			FOR idx:=1 TO nMoverCount DO 
				nMoverInListIndex := nMoverLineDescending[nListCounter, idx];
				IF nMoverInListIndex > 0 THEN
					FOR idx2:=1 TO nMoverCount DO
						IF  MoversToSort[idx2].nMoverIndex > 0
						AND MoversToSort[idx2].nMoverIndex = nMoverInListIndex
						THEN
							IF MoversToSort[idx2].nMoverTrackOID = nTrackOID THEN
								nMoverLineCounter := nMoverLineCounter +1;
								nMoverLineDescend[nMoverLineCounter] := nMoverInListIndex;
							END_IF						
						END_IF
					END_FOR
				END_IF
			END_FOR
			
			nListCounter := nListCounter -1;
		END_WHILE
	


		
	    // Generating the ascending mover line
		FOR idx:=1 TO nMoverLineCounter DO 
			nDescendingCounter := idx;
			nAscendingCounter  := nMoverQueuCounterTotal +1-idx;
		
			IF  nAscendingCounter >  0 
			AND nAscendingCounter <= maxNumMover
			THEN
				nMoverLineAscend[nAscendingCounter] := nMoverLineDescend[nDescendingCounter];	
			ELSE
				nErrorID := -36;	
			END_IF
		END_FOR
		

	
		// Set the needed sorting direction 		
		IF nSortingDirection = eSortingDirection.ascending THEN
			nMoverLineSorted := nMoverLineAscend;
		ELSE
			nMoverLineSorted := nMoverLineDescend;
		END_IF
	
		
	    // Update mover list 
		sMoverSortedInfo := '';
		IF nMoverLineCounter = nMoverCount THEN	
			FOR idx:=1 TO nMoverLineCounter DO 
				nMoverInListIndex := nMoverLineSorted[idx];
				IF nMoverInListIndex > 0 THEN
					FOR idx2:=1 TO nMoverCount DO
						IF MoversToSort[idx2].nMoverIndex = nMoverInListIndex THEN
							MoversSorted[idx] := MoversToSort[idx2];
							 sMoverSortedInfo := CONCAT(sMoverSortedInfo, ' M');
							 sMoverSortedInfo := CONCAT(sMoverSortedInfo, UDINT_TO_STRING(MoversSorted[idx].nMoverIndex));
							EXIT;
						END_IF
					END_FOR
				END_IF		
			END_FOR
		ELSE
			nErrorID := -33;
		END_IF	

	END_IF
	

	CASE nErrorID OF
	  0:// Sorting successfully done	
		MoversList := MoversSorted;
		THIS^.ClearTrackOrder();
		      SortList := UDINT_TO_INT(nMoverLineCounter);    // Returning the number of movers sorted
		sStatusMessage := sMoverSortedInfo;	

	-31: sStatusMessage := 'Sort: No mover in list';
	-32: sStatusMessage := 'Sort: No track specified to sort on';
	-33: sStatusMessage := 'Sort: Mover found on track not specified for sorting';
	-34: sStatusMessage := 'Sort: Sorting origin bigger than length of first track';
	-35: sStatusMessage := 'Sort: Sorting origin was set to negative value';
	-36: sStatusMessage :=  CONCAT('Sort: Sorting impossible, Tracks are not consecutive! Failed at segment: ', UDINT_TO_STRING(nFailedAt));
	-37: sStatusMessage := 'Sort: Sorting not possible, check track order.';
	ELSE
		sStatusMessage := 'Sorting Error';
	END_CASE
	
	IF nErrorID < 0 THEN
		SortList := nErrorID;  // Returning the error code
	END_IF
END_METHOD

END_FUNCTION_BLOCK

// XPlanarStandardFunctions/Station/I_List
INTERFACE I_List EXTENDS __SYSTEM.IQueryInterface

{attribute 'hide'}
{attribute 'obsolete' := 'Obsolete: Please use P_SortingMode instead'}
PROPERTY P_eSortingMode : eSortingMode
GET
END_GET
SET
END_SET
END_PROPERTY

{attribute 'hide'}
{attribute 'obsolete' := 'Obsolete: Please use P_SortingOrigin instead'}
PROPERTY P_fSortingOrigin : LREAL
GET
END_GET
SET
END_SET
END_PROPERTY

{attribute 'hide'}
{attribute 'obsolete' := 'Obsolete: Please use P_NumberInList instead'}
PROPERTY P_nNumberInList : UDINT
GET
END_GET
END_PROPERTY

{attribute 'hide'}
{attribute 'obsolete' := 'Obsolete: Please use P_Result instead'}
PROPERTY P_nResult : DINT
GET
END_GET
END_PROPERTY

{attribute 'hide'}
{attribute 'obsolete' := 'Obsolete: Please use P_SortingMode instead'}
PROPERTY P_nSortingMode : INT
GET
END_GET
SET
END_SET
END_PROPERTY

{attribute 'hide'}
{attribute 'obsolete' := 'Obsolete: Please use P_Message instead'}

PROPERTY P_sMessage : STRING
GET
END_GET
END_PROPERTY

METHOD AddMover : DINT
VAR_INPUT
	ipMover		: I_XPlanarMoverStandard;
END_VAR
END_METHOD

METHOD AddTrack : DINT
VAR_INPUT
	i_Track	: I_TrackStandard;
END_VAR
END_METHOD

METHOD ClearList : BOOL
VAR_INPUT
END_VAR
END_METHOD

METHOD ClearTrackOrder : BOOL
VAR_INPUT
END_VAR
END_METHOD

METHOD GetMoverIndexInListPosition : UDINT
VAR_INPUT
	nListIndex	: UDINT;
END_VAR
END_METHOD

METHOD GetMoverInListPosition : I_XPlanarMoverStandard
VAR_INPUT
	nListPosition	: UDINT;
END_VAR
END_METHOD

PROPERTY P_FirstInList : I_XPlanarMoverStandard
GET
END_GET
END_PROPERTY

PROPERTY P_Message : STRING
GET
END_GET
END_PROPERTY

PROPERTY P_MoverList : REFERENCE TO ARRAY [1..maxNumMover] OF ST_MoverInList
GET
END_GET
END_PROPERTY


PROPERTY P_NumberInList : UDINT
GET
END_GET
END_PROPERTY

PROPERTY P_Result : DINT
GET
END_GET
END_PROPERTY

PROPERTY P_SortingMode : eSortingMode
GET
END_GET
SET
END_SET
END_PROPERTY

PROPERTY P_SortingOrigin : LREAL
GET
END_GET
SET
END_SET
END_PROPERTY

PROPERTY P_TrackBuiltInfo : ST_TrackBuiltInfo
GET
END_GET
SET
END_SET
END_PROPERTY

METHOD RemoveFirstInList : I_XPlanarMoverStandard
VAR_INPUT
END_VAR
END_METHOD

// Removes a mover from the list
METHOD RemoveFromList : DINT
VAR_INPUT
	ipMover			: I_XPlanarMoverStandard;	// Mover to remove
END_VAR
END_METHOD

METHOD SortList : INT
VAR_INPUT
END_VAR
END_METHOD

END_INTERFACE

// XPlanarStandardFunctions/Track/FB_CustomTrackIdTable
FUNCTION_BLOCK FB_CustomTrackIdTable

VAR
	CustomTrackIdTable		: ARRAY [1..Params_XPlanar.maxTrackCount] OF ST_CutomTrackID;
	nTableFillCounter		: UDINT;
END_VAR

METHOD Clear : BOOL
VAR_INPUT
END_VAR


	MEMSET(ADR(CustomTrackIdTable), 0, SIZEOF(CustomTrackIdTable));
		
	Clear := TRUE;
END_METHOD

PROPERTY P_TabelData : ARRAY [1..Params_XPlanar.maxTrackCount] OF ST_CutomTrackID;
GET
P_TabelData := CustomTrackIdTable;
END_GET
END_PROPERTY

METHOD SetTrack : int
VAR_INPUT
	TrackOID	: OTCID;
	nCustomID	: UDINT;	
END_VAR



VAR
	bTrackAlreadIn		: BOOL;
	idx					: UDINT;
END_VAR


	nTableFillCounter := nTableFillCounter +1;
	IF nTableFillCounter <= Params_XPlanar.maxTrackCount THEN
		
		bTrackAlreadIn := FALSE;
		FOR idx:=1 TO Params_XPlanar.maxTrackCount DO
			IF CustomTrackIdTable[idx].TrackOID = TrackOID THEN
				bTrackAlreadIn := TRUE;
			END_IF	
		END_FOR
	
		IF NOT bTrackAlreadIn THEN
			CustomTrackIdTable[nTableFillCounter].nCustomID := nCustomID;
			CustomTrackIdTable[nTableFillCounter].TrackOID  := TrackOID;
			SetTrack := +1;
		ELSE
			SetTrack := -1;
		END_IF
	ELSE
		SetTrack := -2;
	END_IF
END_METHOD

END_FUNCTION_BLOCK

// XPlanarStandardFunctions/Track/FB_TrackStandard
FUNCTION_BLOCK FB_TrackStandard IMPLEMENTS I_TrackStandard 
VAR_INPUT
END_VAR



VAR
	nCustomIndex			: UDINT;
	
	stTrackRef 				: MC_PlanarTrack;
	
	{attribute 'hide'}
	addToGroupCmdFb 		: MC_PlanarFeedback;
	{attribute 'hide'}
	appendLineCmdFb 		: MC_PlanarFeedback;
	{attribute 'hide'}
	appendCircleCmdFb 		: MC_PlanarFeedback;
	{attribute 'hide'}	
	appendPointCmdFb 		: MC_PlanarFeedback;
	{attribute 'hide'}
	clearCmdFb				: MC_PlanarFeedback;
	{attribute 'hide'}
	closeLoopCmdFb			: MC_PlanarFeedback;
	{attribute 'hide'}
	disableCmdFb			: MC_PlanarFeedback;
	{attribute 'hide'}
	enableCmdFb				: MC_PlanarFeedback;
	{attribute 'hide'}
	endAtTrackCmdFb			: MC_PlanarFeedback;
	{attribute 'hide'}
	removeFromGroupCmdFb	: MC_PlanarFeedback;
	{attribute 'hide'}
	startFromTrackCmdFb		: MC_PlanarFeedback;
	{attribute 'hide'}
	resetCmdFb				: MC_PlanarFeedback;
	
	{attribute 'hide'}
	endAtTrackAdvCmdFb		: MC_PlanarFeedback;
	{attribute 'hide'}
	startFromTrackAdvCmdFb	: MC_PlanarFeedback;
	{attribute 'hide'}
	appendLineAdvCmdFb 		: MC_PlanarFeedback;
	{attribute 'hide'}
	appendCircleAdvCmdFb	: MC_PlanarFeedback;
	{attribute 'hide'}
	appendPointAdvCmdFb		: MC_PlanarFeedback;
	
	
	
	stRtAddToGroup 			: ST_CommandReturn;
	stRtAppendLine 			: ST_CommandReturn;
	stRtAppendCircle		: ST_CommandReturn;
	stRtAppendPoint			: ST_CommandReturn;	
	stRtBuildTrack 			: ST_CommandReturn;
	stRtBuildTrackExt 		: ST_CommandReturn;
	stRtBuildTrackAdv 		: ST_CommandReturn;		
	stRtClear				: ST_CommandReturn;
	stRtCloseLoop			: ST_CommandReturn;
	stRtDiable				: ST_CommandReturn;
	stRtEnable				: ST_CommandReturn;
	stRtEndAtTrack			: ST_CommandReturn;
	stRtRemoveFromGroup 	: ST_CommandReturn; 
	stRtStartFromTrack		: ST_CommandReturn;
	stRtReset				: ST_CommandReturn;

	stRtAppendLineAdv 		: ST_CommandReturn;
	stRtAppendCircleAdv		: ST_CommandReturn;
	stRtAppendPointAdv		: ST_CommandReturn;
	stRtEndAtTrackAdv		: ST_CommandReturn;
	stRtStartFromTrackAdv	: ST_CommandReturn;

	

	{attribute 'hide'}
	eState 							: E_MethodKeepAliveTrack;	
	{attribute 'hide'}
	nState							: INT;
	{attribute 'hide'}
	Busy 							: BOOL;
	{attribute 'hide'}
	_bTrackCheck					: BOOL;
	{attribute 'hide'}
	_TrackTableExt					: ARRAY[1..maxNumTrackPoints] OF ST_TrackTable;
	{attribute 'hide'}
	_TrackTableAdv					: ARRAY[1..maxNumTrackPoints] OF ST_TrackTable;
	{attribute 'hide'}
	_TrackTable						: ARRAY [1..maxNumTrackPoints,1..3] OF LREAL;
	//{attribute 'hide'}
	_startFromTrackOptions			: ST_StartFromTrackAdvancedOptions;
	//{attribute 'hide'}
	_endAtTrackOptions				: ST_EndAtTrackAdvancedOptions;
	//{attribute 'hide'}
	_ipStartFromTrack				: I_TrackStandard;	
	//{attribute 'hide'}	
	_ipEndAtTrack 					: I_TrackStandard;
	{attribute 'hide'}
	_bCloseLoop						: BOOL;	
	{attribute 'hide'}
	_nTrackBuilderErrorSituation	: UDINT;
	{attribute 'hide'}
	sBuildTrackExtInfoText			: STRING;
	{attribute 'hide'}
	sBuildTrackAdvInfoText			: STRING;
	{attribute 'hide'}
	nStateBuildTrackAdvanced 		: INT;
	
	// logging
	{attribute 'hide'}
	stTimeZoneInfo 				: TC2_UTILITIES.ST_TimeZoneInformation; //all times are UTC and must be converted to local time zone. if no timezone given only UTC times are avaialbe		
	{attribute 'hide'}
	_eLogSeverity				: TcEventSeverity := TcEventSeverity.VERBOSE;
	{attribute 'hide'}
	stLastCommand				: ST_TrackCommand;	
	aLog						: ARRAY[0..MAX_LAST_LOGS] OF ST_TrackCommandLog;
	
END_VAR


VAR_STAT
	{attribute 'hide'}	
	nTrackBuiltCountInfo	: UDINT;
	{attribute 'hide'}
	nTrackBuiltCount		: UDINT;
	{attribute 'hide'}
	TrackInfo				: ARRAY[1..maxTrackCount] OF ST_TrackInfo;	
	{attribute 'hide'}
	nTrackBuiltTable		: ARRAY[1..maxTrackCount] OF UDINT;
END_VAR

{attribute 'hide'}
METHOD PROTECTED ccl_BuildTrack : BOOL

VAR_INST
	TrackTableInt		: ARRAY [1..maxNumTrackPoints,1..3] OF LREAL;		
	nState				: INT;
	fbR_TrigExecute 	: R_TRIG;
	bCloseLoopFlag		: BOOL;
	nPointIndex			: INT;
	nPointIndexA		: INT;	
	nPointIndexB		: INT;	
	fTestValue			: LREAL;
	idx1, idx2			: INT;
	trackLinePosStart 	: PositionXYC;
	trackLinePosEnd 	: PositionXYC;
END_VAR
CASE nState OF 
	
	0:	// Init
		stRtBuildTrack.Done := FALSE;
		stRtBuildTrack.Busy := TRUE;
		  TrackTableInt := _TrackTable;
	     bCloseLoopFlag := _bCloseLoop;
		    nPointIndex := -1;
		         nState := 100;
	
		
	100: // Building the track
		IF nPointIndex = -1 THEN
			IF _ipStartFromTrack <> 0 THEN
				nState := 110;
			END_IF
			nPointIndex := 0;
		ELSE
			IF nPointIndex < UINT_TO_INT(maxNumTrackPoints-1) THEN
				IF nPointIndex = 0 THEN
					nPointIndex := 1;
				ELSE
					nPointIndex := nPointIndex + 2;
				END_IF
				
				nPointIndexA := nPointIndex;
				nPointIndexB := nPointIndex +1;
				
				fTestValue := 0;
				FOR idx1:=nPointIndexA TO nPointIndexB DO 
					FOR idx2 := 1 TO 3 DO
						fTestValue := fTestValue + _TrackTable[idx1,idx2];	
					END_FOR
				END_FOR
				
				IF fTestValue > 0 THEN
					nState := 120;
				ELSE
					IF _ipEndAtTrack <> 0 THEN
						nPointIndex := UINT_TO_INT(maxNumTrackPoints);
						     nState := 130;
					ELSE
						nPointIndex := UINT_TO_INT(maxNumTrackPoints);
					END_IF
				END_IF
		
			ELSE
				IF bCloseLoopFlag THEN
					nState := 140;
				ELSE
					nState := 200;
				END_IF	
			END_IF
		END_IF
	
	
	110:  // When starting from another track
			IF _ipStartFromTrack <> 0 THEN
			THIS^.StartFromTrack(_ipStartFromTrack);
			nState := 111;
			END_IF
			
	111: 	
			IF startFromTrackCmdFb.Done THEN
				nState := 100;
			END_IF

	120: // Append Line
			trackLinePosStart.SetValuesXYC( _TrackTable[nPointIndexA,1], _TrackTable[nPointIndexA,2], _TrackTable[nPointIndexA,3]);
			trackLinePosEnd.SetValuesXYC(   _TrackTable[nPointIndexB,1], _TrackTable[nPointIndexB,2], _TrackTable[nPointIndexB,3]);
			THIS^.AppendLine(trackLinePosStart,trackLinePosEnd);
			nState := 121;			
			
	121: 
			IF appendLineCmdFb.Done THEN
				nState := 100;
			END_IF	
			
			
	130:  // When ending at another track
			IF _ipEndAtTrack <> 0 THEN
			THIS^.EndAtTrack(_ipEndAtTrack); 
				nState := 131;
			END_IF
			
	131: 
			IF endAtTrackCmdFb.Done THEN
				nState := 100;
			END_IF		
		
	140:  // Closing the track 
			bCloseLoopFlag := FALSE;
			stTrackRef.CloseLoop(closeLoopCmdFb);
			nState := 141;	
			
	141:
			IF closeLoopCmdFb.Done THEN
				nState := 100;
			END_IF
			
			 
	200: 	// MC_Reset Done
			eState 					:= E_MethodKeepAliveTrack.eIdle; 
			nState 					:= 0;
			stRtBuildTrack.Done 	:= TRUE;
			stRtBuildTrack.Busy 	:= FALSE;
			stRtBuildTrack.Active 	:= FALSE;
			ccl_BuildTrack 			:= TRUE;

END_CASE
END_METHOD

//{attribute 'hide'}
METHOD PROTECTED ccl_BuildTrackAdv : BOOL

VAR_INST
	TrackTableInt		: ARRAY[1..maxNumTrackPoints] OF ST_TrackTable;		
	nState				: INT;
	fbR_TrigExecute 	: R_TRIG;
	bCloseLoopFlag		: BOOL;
	nPointIndex			: UINT;

	trackPos 			: PositionXYC;
	trackPosStart 		: PositionXYC;
	trackPosEnd 		: PositionXYC;
	trackPosRef 		: PositionXYC;
	trackPosStartRef 	: PositionXYC;
	trackPosEndRef 		: PositionXYC;	
	trackPosCenter		: PositionXY;

	nErrorId			: UDINT;	
	nErrorSituation		: UDINT;
	
	nTrackOID			: UDINT;

	idx						: UDINT;
	bPreceedingTrackExists	: BOOL;
	bFollowingTrackExists	: BOOL;
	
	bClockWise	: BOOL;
END_VAR


VAR
	stCommand : ST_TrackCommand;
END_VAR
CASE nState OF 
	

	0:	// Init
		stRtBuildTrackAdv.Active := TRUE;
		stRtBuildTrackAdv.Busy   := TRUE;
		stRtBuildTrackAdv.Done   := FALSE;
		
		   TrackTableInt := _TrackTableAdv;
	      bCloseLoopFlag := _bCloseLoop;
		  	    nErrorId := 0;
		 nErrorSituation := 0;
		     nPointIndex := 0;
		          nState := 10;
				 
				 
	10:	// Check if track table is plausible
		IF _bTrackCheck THEN
			nState := 20;
		ELSE
			nErrorSituation := 1;
			nState := 950;
		END_IF			 
				
 
	20: // Check if track is linked to hardware
		nTrackOID := THIS^.P_OID;	
		IF nTrackOID > 0 THEN
			nState := nState + 10;
		ELSE
			nErrorSituation := 8;
			nState := 950;				
		END_IF	
		
		
	30: // Check if the preceding track exists
		bPreceedingTrackExists := FALSE;
		IF _ipStartFromTrack <> 0 THEN	
			FOR idx:=1 TO maxTrackCount DO 
				IF nTrackBuiltTable[idx] = _ipStartFromTrack.P_OID  THEN
					bPreceedingTrackExists := TRUE;
					EXIT;	
				END_IF
			END_FOR
			
			IF bPreceedingTrackExists THEN
				nState := nState + 10;
			ELSE
				nErrorSituation := 9;
				nState := 950;						
			END_IF	
		ELSE
			nState := nState + 10;
		END_IF
		
		
	40: // Check if the following track exists
		bFollowingTrackExists := FALSE;
		IF _ipEndAtTrack <> 0 THEN	
			FOR idx:=1 TO maxTrackCount DO 
				IF nTrackBuiltTable[idx] = _ipEndAtTrack.P_OID  THEN
					bFollowingTrackExists := TRUE;
					EXIT;	
				END_IF
			END_FOR
			
			IF bFollowingTrackExists THEN
				nState := nState + 10;
			ELSE
				nErrorSituation := 10;
				nState := 950;						
			END_IF	
		ELSE
			nState := nState + 10;
		END_IF		
		
		
	50:	nState := 100;
	
	
		 	 
	100: 	// Building the track
			IF nPointIndex = 0 THEN
				nPointIndex := 1;
				IF _ipStartFromTrack <> 0 THEN
					nState := 110;
				END_IF
			ELSE
				IF nPointIndex < maxNumTrackPoints THEN
					
					IF TrackTableInt[nPointIndex].ePointType = E_PointType.Point THEN
						nState := 200;		
					ELSIF TrackTableInt[nPointIndex].ePointType = E_PointType.Line_Start THEN
						nState := 300;
					ELSIF TrackTableInt[nPointIndex].ePointType = E_PointType.Circle_Start THEN
						nState := 400;	
					ELSIF TrackTableInt[nPointIndex].ePointType = E_PointType.none THEN
						nState := 500;	
					END_IF
					
				END_IF
			END_IF
		
	
	110:  // When starting from another track
			IF TrackTableInt[nPointIndex].ReferenceSystem = 0 THEN
				nState := 120;
			ELSE
				nState := 130;
			END_IF	
	
	120:	// Starting from another track without reference system
			IF _ipStartFromTrack <> 0 THEN
			THIS^.StartFromTrack(_ipStartFromTrack);     
				nState := nState +1;
			END_IF
			
	121: 	IF startFromTrackCmdFb.Done THEN
				nState := 100;
			ELSIF startFromTrackCmdFb.Error THEN
				       nErrorId := startFromTrackCmdFb.ErrorId;
				nErrorSituation := 2;
				nState := 950;				
			END_IF	
	
			
	130:	// Starting from another track with reference system
			IF _ipStartFromTrack <> 0 THEN
			THIS^.StartFromTrackAdv(_ipStartFromTrack, _startFromTrackOptions);     
				nState := nState +1;
			END_IF
			
	131: 	
			IF startFromTrackAdvCmdFb.Done THEN
				nState := 100;
			ELSIF startFromTrackAdvCmdFb.Error THEN
				       nErrorId := startFromTrackAdvCmdFb.ErrorId;
				nErrorSituation := 2;
				nState := 950;				
			END_IF
			



	200:	// Append Point
			IF TrackTableInt[nPointIndex].ReferenceSystem = 0 THEN
				nState := 210;
			ELSE
				nState := 220;
			END_IF

			
	210:	// Append Point without reference system
			trackPos.SetValuesXYC(TrackTableInt[nPointIndex].fPointPosition_X, TrackTableInt[nPointIndex].fPointPosition_Y,  TrackTableInt[nPointIndex].fPointOrientation_C);
	
			THIS^.AppendPoint(trackPosRef);
			nPointIndex := nPointIndex +1;
			nState := nState + 11;	
			
	211:	IF appendPointCmdFb.Done THEN
				nState := 100;
			ELSIF appendPointCmdFb.Error THEN
				       nErrorId := appendPointCmdFb.ErrorId;
				nErrorSituation := 3;
				nState := 950;				
			END_IF			
			
			
	220:	// Append Point with reference system
			trackPosRef.SetValuesXYC(TrackTableInt[nPointIndex].fPointPosition_X, TrackTableInt[nPointIndex].fPointPosition_Y,  TrackTableInt[nPointIndex].fPointOrientation_C);
			trackPosRef.ReferenceId := TrackTableInt[nPointIndex].ReferenceSystem;
	
			THIS^.AppendPoint(trackPosRef);
			nPointIndex := nPointIndex +1;
			nState := nState + 11;	
			
	221:	IF appendPointCmdFb.Done THEN
				nState := 100;
			ELSIF appendPointCmdFb.Error THEN
				       nErrorId := appendPointCmdFb.ErrorId;
				nErrorSituation := 3;
				nState := 950;				
			END_IF


			
	300:	// Append Line
			IF TrackTableInt[nPointIndex].ReferenceSystem = 0 THEN
				nState := 310;
			ELSE
				nState := 320;
			END_IF

	310:	// Adding the line without reference system
			trackPosStart.SetValuesXYC(TrackTableInt[nPointIndex].fPointPosition_X, TrackTableInt[nPointIndex].fPointPosition_Y,  TrackTableInt[nPointIndex].fPointOrientation_C);
			trackPosEnd.SetValuesXYC(TrackTableInt[nPointIndex+1].fPointPosition_X, TrackTableInt[nPointIndex+1].fPointPosition_Y,  TrackTableInt[nPointIndex+1].fPointOrientation_C);
			
			THIS^.AppendLine(trackPosStart,trackPosEnd);
			nState := nState + 1;	
			
	311:	IF appendLineCmdFb.Done THEN
				nPointIndex := nPointIndex +2;
				nState := 100;
			ELSIF appendLineCmdFb.Error THEN
				       nErrorId := appendLineCmdFb.ErrorId;
				nErrorSituation := 4;
				nState := 950;				
			END_IF	

			
	320:	// Adding the line with reference system
			trackPosStartRef.SetValuesXYC(TrackTableInt[nPointIndex].fPointPosition_X, TrackTableInt[nPointIndex].fPointPosition_Y,  TrackTableInt[nPointIndex].fPointOrientation_C);
			trackPosEndRef.SetValuesXYC(TrackTableInt[nPointIndex+1].fPointPosition_X, TrackTableInt[nPointIndex+1].fPointPosition_Y,  TrackTableInt[nPointIndex+1].fPointOrientation_C);
			
			trackPosStartRef.ReferenceId := TrackTableInt[nPointIndex].ReferenceSystem;
			trackPosEndRef.ReferenceId   := TrackTableInt[nPointIndex+1].ReferenceSystem;

			THIS^.AppendLine(trackPosStartRef,trackPosEndRef);
			
			nState := nState + 1;	
			
	321:	IF appendLineCmdFb.Done THEN
				nPointIndex := nPointIndex +2;
				nState := 100;
			ELSIF appendLineCmdFb.Error THEN
				       nErrorId := appendLineCmdFb.ErrorId;
				nErrorSituation := 4;
				nState := 950;				
			END_IF		
			

			
	400:	// Append Circle
			IF TrackTableInt[nPointIndex].ReferenceSystem = 0 THEN
				nState := 410;
			ELSE
				nState := 420;
			END_IF
			
	410:	// Append Circle without reference system
			trackPosStart.SetValuesXYC( TrackTableInt[nPointIndex+0].fPointPosition_X,  TrackTableInt[nPointIndex+0].fPointPosition_Y,    TrackTableInt[nPointIndex+0].fPointOrientation_C);
			trackPosCenter.SetValuesXY( TrackTableInt[nPointIndex+1].fPointPosition_X,  TrackTableInt[nPointIndex+1].fPointPosition_Y );
			trackPosEnd.SetValuesXYC(   TrackTableInt[nPointIndex+2].fPointPosition_X,  TrackTableInt[nPointIndex+2].fPointPosition_Y,    TrackTableInt[nPointIndex+2].fPointOrientation_C);
			
			bClockWise := FALSE;
			CASE TrackTableInt[nPointIndex+1].eOption OF
			E_PointOption.Circle_Clockwise: 		bClockWise := TRUE;			
			E_PointOption.Circle_CounterClockwise:	bClockWise := FALSE;		
			END_CASE

			THIS^.AppendCircle(trackPosStart,trackPosCenter,trackPosEnd, bClockWise);
			nPointIndex := nPointIndex +3;
			nState := nState + 10;	
			
	411:	IF appendCircleCmdFb.Done THEN
				nState := 100;
			ELSIF appendCircleCmdFb.Error THEN
				       nErrorId := appendCircleCmdFb.ErrorId;
				nErrorSituation := 5;
				nState := 950;				
			END_IF	


	420:	// Append Circle with reference system
			trackPosStartRef.SetValuesXYC( TrackTableInt[nPointIndex+0].fPointPosition_X,  TrackTableInt[nPointIndex+0].fPointPosition_Y,    TrackTableInt[nPointIndex+0].fPointOrientation_C);
			trackPosCenter.SetValuesXY( TrackTableInt[nPointIndex+1].fPointPosition_X,  TrackTableInt[nPointIndex+1].fPointPosition_Y );
			trackPosEndRef.SetValuesXYC(   TrackTableInt[nPointIndex+2].fPointPosition_X,  TrackTableInt[nPointIndex+2].fPointPosition_Y,    TrackTableInt[nPointIndex+2].fPointOrientation_C);

			trackPosStartRef.ReferenceId := TrackTableInt[nPointIndex].ReferenceSystem;
			trackPosEndRef.ReferenceId   := TrackTableInt[nPointIndex+2].ReferenceSystem;			
			
			bClockWise := FALSE;
			CASE TrackTableInt[nPointIndex+1].eOption OF
			E_PointOption.Circle_Clockwise: 		bClockWise := TRUE;			
			E_PointOption.Circle_CounterClockwise:	bClockWise := FALSE;		
			END_CASE

			THIS^.AppendCircle(trackPosStartRef,trackPosCenter,trackPosEndRef, bClockWise);
			nPointIndex := nPointIndex +3;
			nState := nState + 1;	
			
	421:	
			appendCircleCmdFb.Update();
			IF appendCircleCmdFb.Done THEN
				nState := 100;
			ELSIF appendCircleCmdFb.Error THEN
				       nErrorId := appendCircleCmdFb.ErrorId;
				nErrorSituation := 5;
				nState := 950;				
			END_IF	


			
	500:	// Check if this track is ending on another track  
			IF _ipEndAtTrack <> 0 THEN
				nState := nState + 10;	
			ELSE
				nState := 600;
			END_IF			
			
					
	510:  	// Check if this track has a reference system
			IF TrackTableInt[nPointIndex-1].ReferenceSystem = 1 THEN
				nState := 520;
			ELSE
				nState := 530;
			END_IF				
			

	520:	THIS^.EndAtTrackAdv(_ipEndAtTrack, _endAtTrackOptions); 
			nState := nState + 1;	
		
	521:	IF endAtTrackAdvCmdFb.Done THEN
				nState := 900;
			ELSIF endAtTrackAdvCmdFb.Error THEN
				       nErrorId := endAtTrackAdvCmdFb.ErrorId;
				nErrorSituation := 6;
				nState := 950;				
			END_IF		

			
	530:	THIS^.EndAtTrack(_ipEndAtTrack); 
			nState := nState + 1;	
		
	531:	IF endAtTrackCmdFb.Done THEN
				nState := 900;
			ELSIF endAtTrackCmdFb.Error THEN
				       nErrorId := endAtTrackAdvCmdFb.ErrorId;
				nErrorSituation := 6;
				nState := 950;				
			END_IF					
			
			
	600:	// Check if this track closes the loop
			IF bCloseLoopFlag THEN
				THIS^.CloseLoop();
				nState := nState + 10;
			ELSE
				nState := nState + 100;
			END_IF
			
	610:	IF closeLoopCmdFb.Done THEN
				nState := nState + 90;
			ELSIF closeLoopCmdFb.Error THEN
				       nErrorId := closeLoopCmdFb.ErrorId;
				nErrorSituation := 7;
				nState := 950;				
			END_IF		
			
			
	700:	nState := 900;			
			
				 
	900: 	// BuildTrack successfully done	
			_nTrackBuilderErrorSituation := nErrorSituation;

			nTrackBuiltCount := nTrackBuiltCount +1;
			nTrackBuiltTable[nTrackBuiltCount] := THIS^.P_OID;
				
			stRtBuildTrackAdv.Done 		:= TRUE;
			stRtBuildTrackAdv.Busy 		:= FALSE;
			stRtBuildTrackAdv.Active 	:= FALSE;
			stRtBuildTrackAdv.Error     := FALSE;
			stRtBuildTrackAdv.ErrorID   := nErrorId;
			nState := 1000;
			
			
	950:	// In case of an error
			_nTrackBuilderErrorSituation := nErrorSituation;
 
			stRtBuildTrackAdv.Done 		:= FALSE;
			stRtBuildTrackAdv.Busy 		:= FALSE;
			stRtBuildTrackAdv.Active 	:= FALSE;
			stRtBuildTrackAdv.Error     := TRUE;
			stRtBuildTrackAdv.ErrorID   := nErrorId;
			nState := 1000;
			
			
	1000:	// Done
			CASE _nTrackBuilderErrorSituation OF
			 0:	sBuildTrackAdvInfoText := 'NoError';
			 1:	sBuildTrackAdvInfoText := 'TrackTableNotPlausible';	
			 2:	sBuildTrackAdvInfoText := 'StartFromTrackFailed';	
			 3:	sBuildTrackAdvInfoText := 'AppendPointFailed';
			 4:	sBuildTrackAdvInfoText := 'AppendLineFailed';
			 5:	sBuildTrackAdvInfoText := 'AppendCircleFailed';	
			 6:	sBuildTrackAdvInfoText := 'EndAtTrackFailed';	
			 7:	sBuildTrackAdvInfoText := 'CloseLoopFailed';
			 8:	sBuildTrackAdvInfoText := 'NotLinkedToNC';
			 9: sBuildTrackAdvInfoText := 'Preceeding track needs to be built first!';
			10: sBuildTrackAdvInfoText := 'Following track needs to be built first!';
			END_CASE

			ccl_BuildTrackAdv 	:= TRUE;	
			eState 				:= E_MethodKeepAliveTrack.eIdle; 
			nState 				:= 0;			
			
			
			// Update Command History
			stCommand.eCommandType 				  := eTrackCommand_eBuildTrack;
			stCommand.stBuildTrack.bSuccess 	  := stRtBuildTrackAdv.Done;
			stCommand.stBuildTrack.fTrackLength   := stTrackRef.GetLength();
			stCommand.stBuildTrack.bError 		  := stRtBuildTrackAdv.Error;
			stCommand.stBuildTrack.nErrorCode	  := stRtBuildTrackAdv.ErrorID;
			stCommand.stBuildTrack.sBuildInfoText := sBuildTrackAdvInfoText;
			UpdateCommandHistory(stCommand);

END_CASE

nStateBuildTrackAdvanced := nState;
END_METHOD

//{attribute 'hide'}
METHOD PROTECTED ccl_BuildTrackExt : BOOL

VAR_INST
	TrackTableInt		: ARRAY[1..maxNumTrackPoints] OF ST_TrackTable;;		
	nState				: INT;
	fbR_TrigExecute 	: R_TRIG;
	bCloseLoopFlag		: BOOL;
	nPointIndex			: UINT;

	trackPos 			: PositionXYC;
	trackPosStart 		: PositionXYC;
	trackPosEnd 		: PositionXYC;
	trackPosCenter		: PositionXY;

	nErrorId			: UDINT;	
	nErrorSituation		: UDINT;
	
	nTrackOID			: UDINT;

	idx						: UDINT;
	bPreceedingTrackExists	: BOOL;
	bFollowingTrackExists	: BOOL;
	
	bClockWise	: BOOL;
END_VAR


VAR
	stCommand : ST_TrackCommand;
END_VAR
CASE nState OF 
	

	0:	// Init
		stRtBuildTrackExt.Active := TRUE;
		stRtBuildTrackExt.Busy   := TRUE;
		stRtBuildTrackExt.Done   := FALSE;
		
		   TrackTableInt := _TrackTableExt;
	      bCloseLoopFlag := _bCloseLoop;
		  	    nErrorId := 0;
		 nErrorSituation := 0;
		     nPointIndex := 0;
		          nState := 10;
				 
				 
	10:	// Check if track table is plausible
		IF _bTrackCheck THEN
			nState := 20;
		ELSE
			nErrorSituation := 1;
			nState := 950;
		END_IF			 
				
 
	20: // Check if track is linked to hardware
		nTrackOID := THIS^.P_OID;	
		IF nTrackOID > 0 THEN
			nState := nState + 10;
		ELSE
			nErrorSituation := 8;
			nState := 950;				
		END_IF	
		
		
	30: // Check if the preceding track exists
		bPreceedingTrackExists := FALSE;
		IF _ipStartFromTrack <> 0 THEN	
			FOR idx:=1 TO maxTrackCount DO 
				IF nTrackBuiltTable[idx] = _ipStartFromTrack.P_OID  THEN
					bPreceedingTrackExists := TRUE;
					EXIT;	
				END_IF
			END_FOR
			
			IF bPreceedingTrackExists THEN
				nState := nState + 10;
			ELSE
				nErrorSituation := 9;
				nState := 950;						
			END_IF	
		ELSE
			nState := nState + 10;
		END_IF
		
		
	40: // Check if the following track exists
		bFollowingTrackExists := FALSE;
		IF _ipEndAtTrack <> 0 THEN	
			FOR idx:=1 TO maxTrackCount DO 
				IF nTrackBuiltTable[idx] = _ipEndAtTrack.P_OID  THEN
					bFollowingTrackExists := TRUE;
					EXIT;	
				END_IF
			END_FOR
			
			IF bFollowingTrackExists THEN
				nState := nState + 10;
			ELSE
				nErrorSituation := 10;
				nState := 950;						
			END_IF	
		ELSE
			nState := nState + 10;
		END_IF		
		
		
	50:	nState := 100;
	
	
		 	 
	100: 	// Building the track
			IF nPointIndex = 0 THEN
				IF _ipStartFromTrack <> 0 THEN
					nState := 110;
				END_IF
				nPointIndex := 1;
			ELSE
				IF nPointIndex < maxNumTrackPoints THEN
					
					IF TrackTableInt[nPointIndex].ePointType = E_PointType.Point THEN
						nState := 200;		
					ELSIF TrackTableInt[nPointIndex].ePointType = E_PointType.Line_Start THEN
						nState := 300;
					ELSIF TrackTableInt[nPointIndex].ePointType = E_PointType.Circle_Start THEN
						nState := 400;	
					ELSIF TrackTableInt[nPointIndex].ePointType = E_PointType.none THEN
						nState := 500;	
					END_IF
					
				END_IF
			END_IF
		
	
	110:  // When starting from another track
			IF _ipStartFromTrack <> 0 THEN
			THIS^.StartFromTrack(_ipStartFromTrack);
			nState := 111;
			END_IF
			
	111: 	
			IF startFromTrackCmdFb.Done THEN
				nState := 100;
			ELSIF startFromTrackCmdFb.Error THEN
				       nErrorId := startFromTrackCmdFb.ErrorId;
				nErrorSituation := 2;
				nState := 950;				
			END_IF
			
			
			
	200:	// Append Point
			trackPos.SetValuesXYC(TrackTableInt[nPointIndex].fPointPosition_X, TrackTableInt[nPointIndex].fPointPosition_Y,  TrackTableInt[nPointIndex].fPointOrientation_C);
			THIS^.AppendPoint(trackPos);
			nPointIndex := nPointIndex +1;
			nState := nState + 10;	
			
	210:	IF appendPointCmdFb.Done THEN
				nState := 100;
			ELSIF appendPointCmdFb.Error THEN
				       nErrorId := appendPointCmdFb.ErrorId;
				nErrorSituation := 3;
				nState := 950;				
			END_IF


			
	300:	// Append Line
			trackPosStart.SetValuesXYC(TrackTableInt[nPointIndex].fPointPosition_X, TrackTableInt[nPointIndex].fPointPosition_Y,  TrackTableInt[nPointIndex].fPointOrientation_C);
			trackPosEnd.SetValuesXYC(TrackTableInt[nPointIndex+1].fPointPosition_X, TrackTableInt[nPointIndex+1].fPointPosition_Y,  TrackTableInt[nPointIndex+1].fPointOrientation_C);
			THIS^.AppendLine(trackPosStart,trackPosEnd);
			nPointIndex := nPointIndex +2;
			nState := nState + 10;	
			
	310:	IF appendLineCmdFb.Done THEN
				nState := 100;
			ELSIF appendLineCmdFb.Error THEN
				       nErrorId := appendLineCmdFb.ErrorId;
				nErrorSituation := 4;
				nState := 950;				
			END_IF		
			
			
	400:	// Append Circle
			trackPosStart.SetValuesXYC( TrackTableInt[nPointIndex+0].fPointPosition_X,  TrackTableInt[nPointIndex+0].fPointPosition_Y,    TrackTableInt[nPointIndex+0].fPointOrientation_C);
			trackPosCenter.SetValuesXY( TrackTableInt[nPointIndex+1].fPointPosition_X,  TrackTableInt[nPointIndex+1].fPointPosition_Y );
			trackPosEnd.SetValuesXYC(   TrackTableInt[nPointIndex+2].fPointPosition_X,  TrackTableInt[nPointIndex+2].fPointPosition_Y,    TrackTableInt[nPointIndex+2].fPointOrientation_C);

			bClockWise := FALSE;
			CASE TrackTableInt[nPointIndex+1].eOption OF
			E_PointOption.Circle_Clockwise: 		bClockWise := TRUE;			
			E_PointOption.Circle_CounterClockwise:	bClockWise := FALSE;		
			END_CASE

			THIS^.AppendCircle(trackPosStart,trackPosCenter,trackPosEnd, bClockWise);
			nPointIndex := nPointIndex +3;
			nState := nState + 10;	
			
	410:	IF appendCircleCmdFb.Done THEN
				nState := 100;
			ELSIF appendCircleCmdFb.Error THEN
				       nErrorId := appendCircleCmdFb.ErrorId;
				nErrorSituation := 5;
				nState := 950;				
			END_IF	


	500:	// Check if this track is ending on another track 
			IF _ipEndAtTrack <> 0 THEN
				THIS^.EndAtTrack(_ipEndAtTrack); 
				nState := nState + 10;	
			ELSE
				nState := 600;
			END_IF
	
	510:	IF endAtTrackCmdFb.Done THEN
				nState := 900;
			ELSIF endAtTrackCmdFb.Error THEN
				       nErrorId := endAtTrackCmdFb.ErrorId;
				nErrorSituation := 6;
				nState := 950;				
			END_IF		

			
	600:	// Check if this track closes the loop
			IF bCloseLoopFlag THEN
				THIS^.CloseLoop();
				nState := nState + 10;
			ELSE
				nState := nState + 100;
			END_IF
			
	610:	IF closeLoopCmdFb.Done THEN
				nState := nState + 90;
			ELSIF closeLoopCmdFb.Error THEN
				       nErrorId := closeLoopCmdFb.ErrorId;
				nErrorSituation := 7;
				nState := 950;				
			END_IF		
			
			
	700:	nState := 900;			
			
				 
	900: 	// BuildTrack successfully done	
			_nTrackBuilderErrorSituation := nErrorSituation;

			nTrackBuiltCount := nTrackBuiltCount +1;
			nTrackBuiltTable[nTrackBuiltCount] := THIS^.P_OID;
				
			stRtBuildTrackExt.Done 		:= TRUE;
			stRtBuildTrackExt.Busy 		:= FALSE;
			stRtBuildTrackExt.Active 	:= FALSE;
			stRtBuildTrackExt.Error     := FALSE;
			stRtBuildTrackExt.ErrorID   := nErrorId;
			nState := 1000;
			
			
	950:	// In case of an error
			_nTrackBuilderErrorSituation := nErrorSituation;
 
			stRtBuildTrackExt.Done 		:= FALSE;
			stRtBuildTrackExt.Busy 		:= FALSE;
			stRtBuildTrackExt.Active 	:= FALSE;
			stRtBuildTrackExt.Error     := TRUE;
			stRtBuildTrackExt.ErrorID   := nErrorId;
			nState := 1000;
			
			
	1000:	// Done
			CASE _nTrackBuilderErrorSituation OF
			 0:	sBuildTrackExtInfoText := 'NoError';
			 1:	sBuildTrackExtInfoText := 'TrackTableNotPlausible';	
			 2:	sBuildTrackExtInfoText := 'StartFromTrackFailed';	
			 3:	sBuildTrackExtInfoText := 'AppendPointFailed';
			 4:	sBuildTrackExtInfoText := 'AppendLineFailed';
			 5:	sBuildTrackExtInfoText := 'AppendCircleFailed';	
			 6:	sBuildTrackExtInfoText := 'EndAtTrackFailed';	
			 7:	sBuildTrackExtInfoText := 'CloseLoopFailed';
			 8:	sBuildTrackExtInfoText := 'NotLinkedToNC';
			 9: sBuildTrackExtInfoText := 'Preceeding track needs to be built first!';
			10: sBuildTrackExtInfoText := 'Following track needs to be built first!';
			END_CASE

			ccl_BuildTrackExt 	:= TRUE;	
			eState 				:= E_MethodKeepAliveTrack.eIdle; 
			nState 				:= 0;			
			
			// Update Command History
			stCommand.eCommandType 				  := eTrackCommand_eBuildTrack;
			stCommand.stBuildTrack.bSuccess 	  := stRtBuildTrackExt.Done;
			stCommand.stBuildTrack.fTrackLength   := stTrackRef.GetLength();
			stCommand.stBuildTrack.bError 		  := stRtBuildTrackExt.Error;
			stCommand.stBuildTrack.nErrorCode	  := stRtBuildTrackExt.ErrorID;
			stCommand.stBuildTrack.sBuildInfoText := sBuildTrackExtInfoText;
			UpdateCommandHistory(stCommand);

END_CASE
END_METHOD

{attribute 'hide'}
METHOD PROTECTED ccl_MethodKeepAlive : BOOL
VAR_INPUT
END_VAR
VAR_INST

END_VAR
CASE eState OF
	
	E_MethodKeepAliveTrack.eIdle:
		nState := 0;
	
	E_MethodKeepAliveTrack.eBuildTrack:
		ccl_BuildTrack();	
		
	E_MethodKeepAliveTrack.eBuildTrackExt:
		ccl_BuildTrackExt();	

	E_MethodKeepAliveTrack.eBuildTrackAdv:
		ccl_BuildTrackAdv();					

	E_MethodKeepAliveTrack.eError:
		;
		
END_CASE
END_METHOD

{attribute 'hide'}
METHOD PROTECTED CopyReturnStructure : ST_CommandReturn
VAR_INPUT
	mcInStructur : REFERENCE TO MC_PlanarFeedback;
END_VAR
mcInStructur.Update();
CopyReturnStructure.Active				:= mcInStructur.Active; 
CopyReturnStructure.Busy				:= mcInStructur.Busy;
CopyReturnStructure.Aborted				:= mcInStructur.Aborted;
CopyReturnStructure.Done				:= mcInStructur.Done;
CopyReturnStructure.Error				:= mcInStructur.Error;
CopyReturnStructure.ErrorID 			:= mcInStructur.ErrorId;
CopyReturnStructure.stInfo.nObjectID	:= mcInStructur.objectInfo.Id;
CopyReturnStructure.stInfo.nObjectType	:= mcInStructur.objectInfo.ObjectType;
END_METHOD

PROPERTY ref : PVOID
GET
ref := ADR(stTrackRef);
END_GET
END_PROPERTY

METHOD GetCommandLog : ST_TrackCommandLog
VAR_INPUT
	nNum	: UINT;
END_VAR
GetCommandLog := aLog[nNum];
END_METHOD

METHOD TrackCommandToString : STRING
VAR_INPUT
	eTrackCommand : E_TrackCommandType;
END_VAR
CASE eTrackCommand OF
	eTrackCommand_eEnable:
		TrackCommandToString := 'enable';
	eTrackCommand_eDisable:
		TrackCommandToString := 'disable';
	eTrackCommand_eBuildTrack:
		TrackCommandToString := 'build track';
	eTrackCommand_eAppendPoint:
 		TrackCommandToString := 'append point';		
	eTrackCommand_eAppendLine:
 		TrackCommandToString := 'append line';		
	eTrackCommand_eAppendCircle:
 		TrackCommandToString := 'append circle';
	eTrackCommand_eCloseLoop:
		TrackCommandToString := 'close loop';				
	eTrackCommand_eStartFromTrack:
		TrackCommandToString := 'start from track';
	eTrackCommand_eEndAtTrack:
		TrackCommandToString := 'end at track';
	eTrackCommand_eAddToGroup:
		TrackCommandToString := 'add to group';
	eTrackCommand_eRemoveFromGroup:
		TrackCommandToString := 'remove from group';	
	eTrackCommand_eReset :
		TrackCommandToString := 'reset';	
	
END_CASE
END_METHOD

METHOD UpdateCommandHistory
VAR_IN_OUT 
	stCommand : ST_TrackCommand;
END_VAR
VAR
	lDCTime				: ULINT;
	fbTimeConvert 		: FB_FileTimeToTzSpecificLocalTime; 
	lTzCorrectDCTime 	: ULINT;
	stTrackCommand 		: ST_TrackCommandLog; 
	fbFormatString		: FB_FormatString;
END_VAR

VAR_INST
	fbLoggerArgs	: FB_TcArguments;
	fbSourceInfo 	: FB_TcSourceInfo;
	
	TimeStruct			: DCTIMESTRUCT;
	sDate				: STRING;
	sTime				: STRING;
		
	nCntBuffer			: INT;

END_VAR

// create the timestamp
lDCTime := F_GetActualDcTime64(); 
fbTimeConvert(in:= DCTIME64_TO_FILETIME(lDcTime),tzInfo := stTimeZoneInfo); 
lTzCorrectDCTime:= FILETIME_TO_DCTIME64(fbTimeConvert.out); 
stCommand.stTimeStamp:= DCTIME64_TO_STRING( lTzCorrectDCTime); 


TimeStruct := DCTIME64_TO_DCTIMESTRUCT(lTzCorrectDCTime);

sDate := WORD_TO_STRING(TimeStruct.wYear);
sDate := CONCAT(sDate,'-');
IF TimeStruct.wMonth < 10 THEN sDate := CONCAT(sDate, '0');	END_IF
sDate := CONCAT(sDate,WORD_TO_STRING(TimeStruct.wMonth));
sDate := CONCAT(sDate,'-');
IF TimeStruct.wDay < 10 THEN sDate := CONCAT(sDate, '0');	END_IF
sDate := CONCAT(sDate,WORD_TO_STRING(TimeStruct.wDay));

sTime := '';
IF TimeStruct.wHour < 10 THEN sTime := CONCAT(sTime, '0');	END_IF
sTime := CONCAT(sTime, WORD_TO_STRING(TimeStruct.wHour));
sTime := CONCAT(sTime,':');
IF TimeStruct.wMinute < 10 THEN sTime := CONCAT(sTime, '0');END_IF
sTime := CONCAT(sTime,WORD_TO_STRING(TimeStruct.wMinute));
sTime := CONCAT(sTime,':');
IF TimeStruct.wSecond < 10 THEN sTime := CONCAT(sTime, '0');END_IF
sTime := CONCAT(sTime,WORD_TO_STRING(TimeStruct.wSecond)); 
sTime := CONCAT(sTime,'.');
IF TimeStruct.wMilliseconds < 100 THEN sTime := CONCAT(sTime, '0');END_IF
IF TimeStruct.wMilliseconds <  10 THEN sTime := CONCAT(sTime, '0');END_IF
sTime := CONCAT(sTime,WORD_TO_STRING(TimeStruct.wMilliseconds)); 



CASE _eLogSeverity OF
	
	TcEventSeverity.Critical :;
	
	TcEventSeverity.ERROR:;
	
	TcEventSeverity.INFO:;
	
	TcEventSeverity.VERBOSE:
		
		CASE stCommand.eCommandType OF	

		eTrackCommand_eReset:
			stTrackCommand.sCommandType   := TrackCommandToString(stCommand.eCommandType);
			stTrackCommand.sTimeStamp 	  := stCommand.stTimeStamp;
			stTrackCommand.sTimeStampDate := sDate;
			stTrackCommand.sTimeStampTime := sTime;			
			stTrackCommand.sText          := 'Reset Cmd';

		eTrackCommand_eEnable:
			stTrackCommand.sCommandType   := TrackCommandToString(stCommand.eCommandType);
			stTrackCommand.sTimeStamp 	  := stCommand.stTimeStamp;
			stTrackCommand.sTimeStampDate := sDate;
			stTrackCommand.sTimeStampTime := sTime;		
			stTrackCommand.sText          := 'Enable Cmd';

		eTrackCommand_eDisable:
			stTrackCommand.sCommandType   := TrackCommandToString(stCommand.eCommandType);
			stTrackCommand.sTimeStamp 	  := stCommand.stTimeStamp;
			stTrackCommand.sTimeStampDate := sDate;
			stTrackCommand.sTimeStampTime := sTime;		
			stTrackCommand.sText          := 'Disable Cmd';

		eTrackCommand_eAppendPoint:
			stTrackCommand.sCommandType := TrackCommandToString(stCommand.eCommandType);
			
			fbFormatString.sFormat := 'Pos: X:%.1f;Y:%.1f ';
			fbFormatString.arg1 := F_LREAL(stCommand.stTrackAppendPoint.positionX);
			fbFormatString.arg2 := F_LREAL(stCommand.stTrackAppendPoint.positionY);

			fbFormatString();
			stTrackCommand.sText          := fbFormatString.sOut;
			stTrackCommand.sTimeStamp 	  := stCommand.stTimeStamp;
			stTrackCommand.sTimeStampDate := sDate;
			stTrackCommand.sTimeStampTime := sTime;		
	
		eTrackCommand_eAppendLine:
			stTrackCommand.sCommandType := TrackCommandToString(stCommand.eCommandType);
			
			fbFormatString.sFormat := 'StartPos: X:%.1f;Y:%.1f; EndPos X:%.1f;Y:%.1f';
			fbFormatString.arg1 := F_LREAL(stCommand.stTrackAppendLine.startPositionx);
			fbFormatString.arg2 := F_LREAL(stCommand.stTrackAppendLine.startPositiony);
			fbFormatString.arg3 := F_LREAL(stCommand.stTrackAppendLine.endPositionx);
			fbFormatString.arg4 := F_LREAL(stCommand.stTrackAppendLine.endPositiony);	

			fbFormatString();
			stTrackCommand.sText          := fbFormatString.sOut;
			stTrackCommand.sTimeStamp 	  := stCommand.stTimeStamp;
			stTrackCommand.sTimeStampDate := sDate;
			stTrackCommand.sTimeStampTime := sTime;	
	
		eTrackCommand_eAppendCircle:
			fbFormatString.sFormat := 'StartPos: X:%.1f;Y:%.1f; CenterPos X:%.1f;Y:%.1f EndPos X:%.1f;Y:%.1f';
			fbFormatString.arg1 := F_LREAL(stCommand.stTrackAppendCircle.startPositionX);
			fbFormatString.arg2 := F_LREAL(stCommand.stTrackAppendCircle.startPositionY);
			fbFormatString.arg3 := F_LREAL(stCommand.stTrackAppendCircle.centerPositionX);
			fbFormatString.arg4 := F_LREAL(stCommand.stTrackAppendCircle.centerPositionY);
			fbFormatString.arg5 := F_LREAL(stCommand.stTrackAppendCircle.endPositionX);
			fbFormatString.arg6 := F_LREAL(stCommand.stTrackAppendCircle.endPositionY);
			fbFormatString();
			
			stTrackCommand.sCommandType	  := TrackCommandToString(stCommand.eCommandType);
			stTrackCommand.sText          := fbFormatString.sOut;
			stTrackCommand.sTimeStamp 	  := stCommand.stTimeStamp;
			stTrackCommand.sTimeStampDate := sDate;
			stTrackCommand.sTimeStampTime := sTime;		

		eTrackCommand_eBuildTrack:
			IF stCommand.stBuildTrack.bSuccess THEN
				fbFormatString.sFormat := 'Track Length: %.1f';
				fbFormatString.arg1    := F_LREAL(stCommand.stBuildTrack.fTrackLength);
				fbFormatString();
				stTrackCommand.sText   := fbFormatString.sOut;
			ELSIF stCommand.stBuildTrack.bError THEN
				IF stCommand.stBuildTrack.nErrorCode > 0 THEN			
					fbFormatString.sFormat := 'Error Code: %d';
					fbFormatString.arg1    := F_UDINT(stCommand.stBuildTrack.nErrorCode);	
					fbFormatString();
					stTrackCommand.sText   := fbFormatString.sOut;
				ELSE
					stTrackCommand.sText := stCommand.stBuildTrack.sBuildInfoText;
				END_IF
			ELSE							
				stTrackCommand.sText   :='Error - Check Track-Initialization';
			END_IF
			
			stTrackCommand.sCommandType   := TrackCommandToString(stCommand.eCommandType);		
			stTrackCommand.sTimeStamp 	  := stCommand.stTimeStamp;
			stTrackCommand.sTimeStampDate := sDate;
			stTrackCommand.sTimeStampTime := sTime;				

		eTrackCommand_eStartFromTrack:		
			stTrackCommand.sCommandType   := TrackCommandToString(stCommand.eCommandType);
			fbFormatString.sFormat 		  := 'Start from Track OID: %d ';
			fbFormatString.arg1 		  := F_UDINT(stCommand.ststartfromTrack.nTrackOID);
			fbFormatString();
			stTrackCommand.sText          := fbFormatString.sOut;
			stTrackCommand.sTimeStamp     := stCommand.stTimeStamp;
			stTrackCommand.sTimeStampDate := sDate;
			stTrackCommand.sTimeStampTime := sTime;		
						
		eTrackCommand_eEndAtTrack:		
			stTrackCommand.sCommandType   := TrackCommandToString(stCommand.eCommandType);
			fbFormatString.sFormat 		  := 'End at Track OID: %d ';
			fbFormatString.arg1 		  := F_UDINT(stCommand.stEndAtTrack.nTrackOID);
			fbFormatString();
			stTrackCommand.sText          := fbFormatString.sOut;
			stTrackCommand.sTimeStamp     := stCommand.stTimeStamp;
			stTrackCommand.sTimeStampDate := sDate;
			stTrackCommand.sTimeStampTime := sTime;		
			
		eTrackCommand_eCloseLoop:
			stTrackCommand.sCommandType   := TrackCommandToString(stCommand.eCommandType);			
			stTrackCommand.sText          := 'Close Loop Cmd';
			stTrackCommand.sTimeStamp     := stCommand.stTimeStamp;
			stTrackCommand.sTimeStampDate := sDate;
			stTrackCommand.sTimeStampTime := sTime;		

		eTrackCommand_eAddToGroup:
			stTrackCommand.sCommandType := TrackCommandToString(stCommand.eCommandType);
						
			stTrackCommand.sText          := 'Add to Group Cmd';
			stTrackCommand.sTimeStamp     := stCommand.stTimeStamp;	
			stTrackCommand.sTimeStampDate := sDate;
			stTrackCommand.sTimeStampTime := sTime;			
			

		eTrackCommand_eRemoveFromGroup:
			stTrackCommand.sCommandType := TrackCommandToString(stCommand.eCommandType);
			stTrackCommand.sText          := 'Remove from Group Cmd';
			stTrackCommand.sTimeStamp     := stCommand.stTimeStamp;	
			stTrackCommand.sTimeStampDate := sDate;
			stTrackCommand.sTimeStampTime := sTime;						
		
		END_CASE
		
		
	TcEventSeverity.WARNING:;

END_CASE


aLog[0] :=  stTrackCommand;
FOR nCntBuffer := UINT_TO_INT(MAX_LAST_LOGS) TO 1  BY -1 DO
	MEMCPY(destAddr:=ADR(aLog[nCntBuffer]) , srcAddr:=ADR(aLog[nCntBuffer-1]) , n:=SIZEOF(ST_TrackCommandLog) );
	aLog[nCntBuffer].nNo := nCntBuffer;
	MEMSET(destAddr:=ADR(aLog[nCntBuffer-1]) , fillByte:=0 , n:= SIZEOF(ST_TrackCommandLog));
END_FOR
END_METHOD

PROPERTY P_AddToGroup : REFERENCE TO ST_CommandReturn
GET
P_AddToGroup REF= stRtAddToGroup;
END_GET
END_PROPERTY

PROPERTY P_AppendCircle : REFERENCE TO ST_CommandReturn
GET
P_AppendCircle REF= stRtAppendCircle;
END_GET
END_PROPERTY

PROPERTY P_AppendLine : REFERENCE TO ST_CommandReturn
GET
P_AppendLine REF= stRtAppendLine;
END_GET
END_PROPERTY

PROPERTY P_AppendPoint : REFERENCE TO ST_CommandReturn
GET
P_AppendPoint REF= stRtAppendPoint;
END_GET
END_PROPERTY

{attribute 'hide'}
PROPERTY P_BuildTrack : REFERENCE TO ST_CommandReturn
GET
P_BuildTrack REF= stRtBuildTrack;
END_GET
END_PROPERTY

PROPERTY P_BuildTrackAdvanced : REFERENCE TO ST_CommandReturn
GET
P_BuildTrackAdvanced REF= stRtBuildTrackAdv;
END_GET
END_PROPERTY

PROPERTY P_BuildTrackAdvanced_Check : int
GET
P_BuildTrackAdvanced_Check := nStateBuildTrackAdvanced;
END_GET
END_PROPERTY

PROPERTY P_BuildTrackAdvancedInfoText : STRING
GET

P_BuildTrackAdvancedInfoText := sBuildTrackAdvInfoText;
END_GET
END_PROPERTY

PROPERTY P_BuildTrackExt : REFERENCE TO ST_CommandReturn
GET
P_BuildTrackExt REF= stRtBuildTrackExt;
END_GET
END_PROPERTY

PROPERTY P_BuildTrackExtInfoText : STRING
GET

P_BuildTrackExtInfoText := sBuildTrackExtInfoText;
END_GET
END_PROPERTY

PROPERTY P_Clear : REFERENCE TO ST_CommandReturn
GET
P_Clear REF= stRtClear;
END_GET
END_PROPERTY

PROPERTY P_CloseLoop : REFERENCE TO ST_CommandReturn
GET
P_CloseLoop REF= stRtCloseLoop;
END_GET
END_PROPERTY

PROPERTY P_Disable : REFERENCE TO ST_CommandReturn
GET
P_Disable REF= stRtDiable;
END_GET
END_PROPERTY

PROPERTY P_Enable : REFERENCE TO ST_CommandReturn
GET
P_Enable REF= stRtEnable;
END_GET
END_PROPERTY

PROPERTY P_EndAtTrack : REFERENCE TO ST_CommandReturn
GET
P_EndAtTrack REF= stRtEndAtTrack;
END_GET
END_PROPERTY

PROPERTY P_RemoveFromGroup : REFERENCE TO ST_CommandReturn
GET
P_RemoveFromGroup REF= stRtRemoveFromGroup;
END_GET
END_PROPERTY

PROPERTY P_Reset : REFERENCE TO ST_CommandReturn
GET
P_Reset REF= stRtReset;
END_GET
END_PROPERTY

PROPERTY P_StartFromTrack : REFERENCE TO ST_CommandReturn
GET
P_StartFromTrack REF= stRtStartFromTrack;
END_GET
END_PROPERTY

METHOD AddToGroup : BOOL
VAR_INPUT
	group : REFERENCE TO MC_PlanarGroup;
END_VAR



VAR
	stCommand 	: ST_TrackCommand;
	sText		: STRING;
END_VAR

MEMSET(ADR(stRtAddToGroup), 0, SIZEOF(stRtAddToGroup));

stTrackRef.AddToGroup(addToGroupCmdFb, group);
AddToGroup := True;




// Update Command History
sText := 'Group OID: ';
sText := CONCAT(sText, UDINT_TO_STRING(group.MCTOPLC_STD.GroupOID));

stCommand.eCommandType := eTrackCommand_eAddToGroup;
stCommand.sText        := sText;

UpdateCommandHistory(stCommand);
END_METHOD

METHOD AppendCircle : BOOL
VAR_INPUT
	startPosition	: REFERENCE TO PositionXYC;
	centerPosition	: REFERENCE TO PositionXY;
	endPosition 	: REFERENCE TO PositionXYC;
	clockwise		: REFERENCE TO BOOL;
END_VAR




VAR
	stCommand : ST_TrackCommand;
END_VAR
IF NOT Busy THEN
	MEMSET(ADR(stRtAppendCircle), 0, SIZEOF(stRtAppendCircle));
	stTrackRef.AppendCircle(appendCircleCmdFb, startPosition, endPosition, centerPosition, clockwise);
	
	AppendCircle := TRUE;
ELSE
	AppendCircle := FALSE;
END_IF



// Update Command History
stCommand.stTrackAppendCircle.startPositionx  := startPosition.x;
stCommand.stTrackAppendCircle.startPositiony  := startPosition.y;
stCommand.stTrackAppendCircle.centerPositionX := centerPosition.x;
stCommand.stTrackAppendCircle.centerPositionY := centerPosition.y;
stCommand.stTrackAppendCircle.endPositionx    := endPosition.x;
stCommand.stTrackAppendCircle.endPositiony    := endPosition.y;

stCommand.eCommandType := eTrackCommand_eAppendCircle;
UpdateCommandHistory(stCommand);
END_METHOD

METHOD AppendLine : BOOL
VAR_INPUT
	startPosition	: REFERENCE TO PositionXYC;
	endPosition 	: REFERENCE TO PositionXYC;
END_VAR




VAR
	stCommand : ST_TrackCommand;
END_VAR
IF NOT Busy THEN
	MEMSET(ADR(stRtAppendLine), 0, SIZEOF(stRtAppendLine));
	stTrackRef.AppendLine(appendLineCmdFb, startPosition, endPosition);
	AppendLine := TRUE;
ELSE
	AppendLine := FALSE;
END_IF


// Update Command History
stCommand.stTrackAppendLine.startPositionx := startPosition.x;
stCommand.stTrackAppendLine.startPositiony := startPosition.y;
stCommand.stTrackAppendLine.endPositionx   := endPosition.x;
stCommand.stTrackAppendLine.endPositiony   := endPosition.y;

stCommand.eCommandType := eTrackCommand_eAppendLine;
UpdateCommandHistory(stCommand);
END_METHOD

METHOD AppendPoint : BOOL
VAR_INPUT
	position	: REFERENCE TO PositionXYC;
END_VAR




VAR
	stCommand : ST_TrackCommand;
END_VAR
IF NOT Busy THEN	
	MEMSET(ADR(stRtAppendPoint), 0, SIZEOF(stRtAppendPoint));
	stTrackRef.AppendPosition(appendPointCmdFb, position);
	
	AppendPoint := TRUE;
ELSE
	AppendPoint := FALSE;
END_IF



// Update Command History 
stCommand.stTrackAppendPoint.positionX := position.x;
stCommand.stTrackAppendPoint.positionY := position.y;
stCommand.eCommandType := eTrackCommand_eAppendPoint;
UpdateCommandHistory(stCommand);
END_METHOD

{attribute 'hide'}
METHOD BuildTrack : BOOL
VAR_INPUT
	TrackTable			: ARRAY [1..maxNumTrackPoints,1..3] OF LREAL;
	ipStartFromTrack	: I_TrackStandard;		
	ipEndAtTrack 		: I_TrackStandard;
	bCloseLoop			: BOOL;
END_VAR


VAR_INST
	TrackTableInt	: ARRAY [1..maxNumTrackPoints,1..3] OF LREAL;		
	
	nState			: INT;
	fbR_TrigExecute : R_TRIG;
	
	bCloseLoopFlag	: BOOL;
	nPointIndex		: INT;
	nPointIndexA	: INT;	
	nPointIndexB	: INT;	
	fTestValue		: LREAL;
	idx1, idx2		: INT;
	
	
	trackLinePosStart 	: PositionXYC;
	trackLinePosEnd 	: PositionXYC;
	
	
END_VAR


VAR
	stCommand 	: ST_TrackCommand;
END_VAR
_TrackTable 		:= TrackTable;		
_ipStartFromTrack 	:= ipStartFromTrack;
_ipEndAtTrack 		:= ipEndAtTrack;
_bCloseLoop 		:= bCloseLoop;	

eState :=  E_MethodKeepAliveTrack.eBuildTrack; 

BuildTrack := TRUE;
END_METHOD

METHOD BuildTrackAdvanced : BOOL
VAR_INPUT
	TrackTable			: REFERENCE TO FB_TrackTableAdvanced;
END_VAR



VAR
	stCommand : ST_TrackCommand;
END_VAR
IF TrackTable.CheckTrackTable() <> 0 THEN
	_bTrackCheck        	:= TrackTable.P_TrackTableCheckResult;
	_TrackTableAdv 			:= TrackTable.P_Table;		
	_ipStartFromTrack 		:= TrackTable.P_StartFromTrack;
	_startFromTrackOptions 	:= TrackTable.P_StartFromTrackOptions;
	_ipEndAtTrack 			:= TrackTable.P_EndAtTrack;
	_endAtTrackOptions 		:= TrackTable.P_EndAtTrackOptions;
	_bCloseLoop 			:= TrackTable.P_CloseTheLoop;	
	
	
	nTrackBuiltCountInfo := nTrackBuiltCountInfo +1;
	TrackInfo[nTrackBuiltCountInfo].TrackOID	   := THIS^.P_OID;
	TrackInfo[nTrackBuiltCountInfo].StartFromTrack := _ipStartFromTrack;
	TrackInfo[nTrackBuiltCountInfo].EndAtTrack	   := _ipStartFromTrack;
	
	MEMSET(ADR(stRtBuildTrackAdv), 0, SIZEOF(stRtBuildTrackAdv));
	
 	eState := E_MethodKeepAliveTrack.eBuildTrackAdv; 

	BuildTrackAdvanced := TRUE;
END_IF
END_METHOD

METHOD BuildTrackExt : BOOL
VAR_INPUT
	TrackTable			: REFERENCE TO FB_TrackTable;
END_VAR



VAR
	stCommand : ST_TrackCommand;
END_VAR
IF TrackTable.CheckTrackTable() <> 0 THEN
	_bTrackCheck        := TrackTable.P_TrackTableCheckResult;
	_TrackTableExt 		:= TrackTable.P_Table;		
	_ipStartFromTrack 	:= TrackTable.P_StartFromTrack;
	_ipEndAtTrack 		:= TrackTable.P_EndAtTrack;
	_bCloseLoop 		:= TrackTable.P_CloseTheLoop;	

	
	nTrackBuiltCountInfo := nTrackBuiltCountInfo +1;
	TrackInfo[nTrackBuiltCountInfo].TrackOID	   := THIS^.P_OID;
	TrackInfo[nTrackBuiltCountInfo].StartFromTrack := _ipStartFromTrack;
	TrackInfo[nTrackBuiltCountInfo].EndAtTrack	   := _ipStartFromTrack;
	
	MEMSET(ADR(stRtBuildTrackExt), 0, SIZEOF(stRtBuildTrackExt));
	
 	eState := E_MethodKeepAliveTrack.eBuildTrackExt; 

	BuildTrackExt := TRUE;
END_IF
END_METHOD

METHOD Clear : BOOL
VAR_INPUT
END_VAR


VAR
	stCommand : ST_TrackCommand;
END_VAR

IF NOT Busy THEN
	MEMSET(ADR(stRtClear), 0, SIZEOF(stRtClear));
	
	MEMSET(ADR(nTrackBuiltTable), 0, SIZEOF(nTrackBuiltTable));
	
	nTrackBuiltCount	 := 0;
	nTrackBuiltCountInfo := 0;
	
	stTrackRef.Clear(clearCmdFb);
	
	Clear := TRUE;
END_IF



// Update Command History
stCommand.eCommandType := eTrackCommand_eClear;
UpdateCommandHistory(stCommand);
END_METHOD

METHOD CloseLoop : BOOL
VAR_INPUT
END_VAR

VAR
	stCommand : ST_TrackCommand;
END_VAR
IF NOT Busy THEN
	MEMSET(ADR(stRtCloseLoop), 0, SIZEOF(stRtCloseLoop));
	stTrackRef.CloseLoop(closeLoopCmdFb);
END_IF
 


// Update Command History
stCommand.eCommandType := eTrackCommand_eCloseLoop;
UpdateCommandHistory(stCommand);
END_METHOD

METHOD cycle : BOOL
VAR_INPUT
END_VAR
stTrackRef.Update();
ccl_MethodKeepAlive();

stRtAddToGroup 			:= CopyReturnStructure(addToGroupCmdFb);
stRtAppendLine 			:= CopyReturnStructure(appendLineCmdFb);
stRtAppendLineAdv 		:= CopyReturnStructure(appendLineAdvCmdFb);
stRtAppendCircle 		:= CopyReturnStructure(appendCircleCmdFb);
stRtAppendCircleAdv 	:= CopyReturnStructure(appendCircleAdvCmdFb);
stRtAppendPoint 		:= CopyReturnStructure(appendPointCmdFb);
stRtAppendPointAdv 		:= CopyReturnStructure(appendPointAdvCmdFb);
stRtClear				:= CopyReturnStructure(clearCmdFb);		
stRtCloseLoop			:= CopyReturnStructure(closeLoopCmdFb);		
stRtDiable				:= CopyReturnStructure(disableCmdFb);		
stRtEnable				:= CopyReturnStructure(enableCmdFb);			
stRtEndAtTrack			:= CopyReturnStructure(endAtTrackCmdFb);	
stRtEndAtTrackAdv		:= CopyReturnStructure(endAtTrackAdvCmdFb);		
stRtRemoveFromGroup 	:= CopyReturnStructure(removeFromGroupCmdFb);
stRtStartFromTrack		:= CopyReturnStructure(startFromTrackCmdFb);
stRtStartFromTrackAdv	:= CopyReturnStructure(startFromTrackAdvCmdFb);
stRtReset				:= CopyReturnStructure(resetCmdFb);
END_METHOD

METHOD Disable : BOOL
VAR_INPUT
END_VAR


VAR
	stCommand : ST_TrackCommand;
END_VAR
IF NOT Busy THEN
	MEMSET(ADR(stRtDiable), 0, SIZEOF(stRtDiable));
	stTrackRef.Disable(disableCmdFb);
	Disable := True;
END_IF




// Update Command History
stCommand.eCommandType := eTrackCommand_eDisable;
UpdateCommandHistory(stCommand);
END_METHOD

METHOD Enable : BOOL
VAR_INPUT
END_VAR


VAR
	stCommand : ST_TrackCommand;
END_VAR

IF NOT Busy THEN
	MEMSET(ADR(stRtEnable), 0, SIZEOF(stRtEnable));
	stTrackRef.Enable(enableCmdFb);
	
	Enable := TRUE;
END_IF



// Update Command History
stCommand.eCommandType := eTrackCommand_eEnable;
UpdateCommandHistory(stCommand);
END_METHOD

METHOD EndAtTrack : BOOL
VAR_INPUT
	ipTrackExt : I_TrackStandard;
END_VAR


VAR
	stCommand : ST_TrackCommand;
	ref : POINTER TO MC_PlanarTrack;
END_VAR
ref := ipTrackExt.ref;
IF NOT Busy THEN
	MEMSET(ADR(stRtEndAtTrack), 0, SIZEOF(stRtEndAtTrack));
	stTrackRef.EndAtTrack(endAtTrackCmdFB, ref^);
	EndAtTrack := TRUE;
ELSE
	EndAtTrack := FALSE;
END_IF




// Update Command History
stCommand.eCommandType 			 := eTrackCommand_eEndAtTrack;
stCommand.stEndAtTrack.nTrackOID := ipTrackExt.P_OID;

UpdateCommandHistory(stCommand);
END_METHOD

{attribute 'hide'}
METHOD EndAtTrackAdv : BOOL
VAR_INPUT
	ipTrackExt : I_TrackStandard;
	endAtOpt	: ST_EndAtTrackAdvancedOptions;
END_VAR


VAR
	stCommand : ST_TrackCommand;
	trackRef  : POINTER TO MC_PlanarTrack;
END_VAR
trackRef := ipTrackExt.ref;
IF NOT Busy THEN
	MEMSET(ADR(stRtEndAtTrackAdv), 0, SIZEOF(stRtEndAtTrackAdv));
	stTrackRef.EndAtTrackAdvanced(endAtTrackAdvCmdFB, trackRef^, endAtOpt);
	EndAtTrackAdv := TRUE;
ELSE
	EndAtTrackAdv := FALSE;
END_IF




// Update Command History
stCommand.eCommandType 			 := eTrackCommand_eEndAtTrack;
stCommand.stEndAtTrack.nTrackOID := ipTrackExt.P_OID;
UpdateCommandHistory(stCommand);
END_METHOD

METHOD GetLength : LREAL;
VAR_INPUT
END_VAR
GetLength := stTrackRef.GetLength();
END_METHOD

METHOD GetMoverPositionAt : BOOL

VAR_INPUT
	(* Arc length value where the position is evaluated. *)
	arcLength : LREAL;
END_VAR
VAR_IN_OUT
	(* The position at the specified arc parameter. *)
	position : PositionXYC;
END_VAR
stTrackRef.GetPositionAt(arcLength, position);
END_METHOD

METHOD GetTrackPositionAt : LREAL
VAR_INPUT
	Position : REFERENCE TO PositionXYC;
END_VAR



VAR_INST
	
	fTest : LREAL;

END_VAR

fTest := stTrackRef.GetArcLengthClosestTo(Position);


GetTrackPositionAt := stTrackRef.GetArcLengthClosestTo(Position);
END_METHOD

METHOD GetTrackPositionAt_XY : LREAL
VAR_INPUT
	x	: LREAL;
	y	: LREAL;
END_VAR



VAR_INST
	
	fTest 		: LREAL;
	posXYC		: PositionXYC;

END_VAR



posXYC.SetValuesXYC(x, y, 0.0);
					
fTest := stTrackRef.GetArcLengthClosestTo(posXYC);			
			
GetTrackPositionAt_XY := stTrackRef.GetArcLengthClosestTo(posXYC);
END_METHOD

PROPERTY P_GroupOID : UDINT
GET


P_GroupOID := stTrackRef.MCTOPLC_STD.GroupOID;
END_GET
END_PROPERTY

PROPERTY P_Info : PlanarObjectInfo
GET
VAR
	


	Info : PlanarObjectInfo;



END_VAR


Info := stTrackRef.GetPlanarObjectInfo();

P_Info := Info;
END_GET
END_PROPERTY

PROPERTY P_MoverCountOnTrack : UDINT
GET
P_MoverCountOnTrack := stTrackRef.MCTOPLC_STD.MoverCountOnTrack;
END_GET
END_PROPERTY

PROPERTY P_MovingMoverCount : UDINT
GET
P_MovingMoverCount := stTrackRef.MCTOPLC_STD.MovingMoverCount;
END_GET
END_PROPERTY

PROPERTY P_OID : UDINT
GET


P_OID := stTrackRef.MCTOPLC_STD.TrackOID;
END_GET
END_PROPERTY

PROPERTY P_OperationMode : MC_PLANAR_TRACK_OPERATION_MODE
GET
P_OperationMode := stTrackRef.MCTOPLC_STD.OperationMode;
END_GET
END_PROPERTY

PROPERTY P_State : MC_PLANAR_STATE
GET
P_State := stTrackRef.MCTOPLC_STD.State;
END_GET
END_PROPERTY

PROPERTY P_TrackBuiltInfo : ST_TrackBuiltInfo
GET
VAR
	
	TrackBuiltInfoTemp : ST_TrackBuiltInfo;

END_VAR


	TrackBuiltInfoTemp.nTrackBuiltCountInfo := nTrackBuiltCountInfo;
	TrackBuiltInfoTemp.TrackInfo 			:= TrackInfo;


	P_TrackBuiltInfo := TrackBuiltInfoTemp;
END_GET
END_PROPERTY

PROPERTY P_TrackRef : POINTER TO MC_PlanarTrack
GET
P_TrackRef := ADR(stTrackRef);
END_GET
END_PROPERTY

METHOD RemoveFromGroup : BOOL
VAR_INPUT
END_VAR




VAR
	stCommand : ST_TrackCommand;
END_VAR
MEMSET(ADR(stRtRemoveFromGroup), 0, SIZEOF(stRtRemoveFromGroup));
stTrackRef.RemoveFromGroup(removeFromGroupCmdFb);
RemoveFromGroup := TRUE;


// Update Command History
stCommand.eCommandType := eTrackCommand_eRemoveFromGroup;
UpdateCommandHistory(stCommand);
END_METHOD

METHOD Reset : BOOL
VAR_INPUT
END_VAR

VAR
	stCommand : ST_TrackCommand;
END_VAR

IF NOT Busy THEN
	MEMSET(ADR(stRtReset), 0, SIZEOF(stRtReset));
	stTrackRef.Reset(resetCmdFb);
	Reset := TRUE;
END_IF


// Update Command History
stCommand.eCommandType := eTrackCommand_eReset;
UpdateCommandHistory(stCommand);
END_METHOD

METHOD StartFromTrack : BOOL
VAR_INPUT
	ipTrackExt : I_TrackStandard;
END_VAR



VAR
	stCommand : ST_TrackCommand;
	ref : POINTER TO MC_PlanarTrack;
END_VAR
ref := ipTrackExt.ref;
IF NOT Busy THEN
	MEMSET(ADR(stRtStartFromTrack), 0, SIZEOF(stRtStartFromTrack));
	stTrackRef.StartFromTrack(startFromTrackCmdFB, ref^);
	StartFromTrack := TRUE;
ELSE
	StartFromTrack := FALSE;
END_IF



// Update Command History
stCommand.eCommandType 				 := eTrackCommand_eStartFromTrack;
stCommand.stStartFromTrack.nTrackOID := ipTrackExt.P_OID;
UpdateCommandHistory(stCommand);
END_METHOD

{attribute 'hide'}
METHOD StartFromTrackAdv : BOOL
VAR_INPUT
	ipTrackExt 		: I_TrackStandard;
	startFromOpt	: ST_StartFromTrackAdvancedOptions;
END_VAR



VAR_INST
	      stCommand : ST_TrackCommand;
	     _trackRef  : POINTER TO MC_PlanarTrack;
	_startFromOpt	: ST_StartFromTrackAdvancedOptions;
END_VAR
_trackRef := ipTrackExt.ref;
_startFromOpt := startFromOpt;


IF NOT Busy THEN
	MEMSET(ADR(stRtStartFromTrackAdv), 0, SIZEOF(stRtStartFromTrackAdv));
	stTrackRef.StartFromTrackAdvanced(startFromTrackAdvCmdFB, _trackRef^, _startFromOpt);
	StartFromTrackAdv := TRUE;
ELSE
	StartFromTrackAdv := FALSE;
END_IF



// Update Command History
stCommand.eCommandType 				 := eTrackCommand_eStartFromTrackAdv;
stCommand.stStartFromTrack.nTrackOID := ipTrackExt.P_OID;
UpdateCommandHistory(stCommand);
END_METHOD

END_FUNCTION_BLOCK

// XPlanarStandardFunctions/Track/I_CustomTrackIndexTable
INTERFACE I_CustomTrackIndexTable

PROPERTY P_TabelData : BOOL
GET
END_GET
END_PROPERTY

END_INTERFACE

// XPlanarStandardFunctions/Visualization/FB_XPlanarVisuDiag
FUNCTION_BLOCK FB_XPlanarVisuDiag
VAR
	aMover 		: ARRAY [1..maxNumMover] OF I_XPlanarMoverStandard;	
	aTrack 		: ARRAY [1..maxTrackCount] OF I_TrackStandard;
END_VAR

METHOD Cycle : BOOL
VAR_INPUT
END_VAR

VAR
	nForCounter : int;
END_VAR


VAR_INST
	
	// Mover log
	nMaxMoverIdtoDisplay 	: INT := 10;
	rtNextMover				: R_TRIG;
	rtPreviousMover			: R_TRIG;


	// Track log	
	nMaxTrackIdtoDisplay 	: INT := 10;
	rtNextTrack				: R_TRIG;
	rtPreviousTrack			: R_TRIG;
		
END_VAR


// Mover
UpdateMoverStatus();

    rtNextMover( CLK := GVL_internal.bNextMover);		
rtPreviousMover( CLK := GVL_internal.bPreviousMover);		    	

IF (     rtPreviousMover.Q 
     AND GVL_internal.nMoverIdToDisplay > 1)
THEN
	GVL_internal.nMoverIdToDisplay := GVL_internal.nMoverIdToDisplay -1;
END_IF

IF  rtNextMover.Q 
AND GVL_internal.nMoverIdToDisplay < UDINT_TO_INT(Params_XPlanar.moverCount)
THEN
	IF aMover[GVL_internal.nMoverIdToDisplay +1] <> 0 THEN
		GVL_internal.nMoverIdToDisplay := GVL_internal.nMoverIdToDisplay + 1;
	END_IF
END_IF



// Track
UpdateTrackLog();

    rtNextTrack( CLK := GVL_internal.bNextTrack);		
rtPreviousTrack( CLK := GVL_internal.bPreviousTrack);		    	

IF  rtPreviousTrack.Q 
AND GVL_internal.nTrackIdToDisplay > 1
THEN
	GVL_internal.nTrackIdToDisplay := GVL_internal.nTrackIdToDisplay -1;
END_IF

IF (rtNextTrack.Q 
AND GVL_internal.nTrackIdToDisplay < UDINT_TO_INT(Params_XPlanar.maxTrackCount))
THEN
	IF aTrack[GVL_internal.nTrackIdToDisplay +1] <> 0 THEN
		GVL_internal.nTrackIdToDisplay := GVL_internal.nTrackIdToDisplay + 1;
	END_IF
END_IF
END_METHOD

METHOD SetStandardMover : BOOL
VAR_INPUT
	ipMover	: I_XPlanarMoverStandard;
	nNum	: UDINT;
END_VAR
IF nNum <= maxNumMover THEN
	aMover[nNum] := ipMover;
END_IF

SetStandardMover := TRUE;
END_METHOD

METHOD SetStandardTrack : BOOL
VAR_INPUT
	ipTrack	: I_TrackStandard;
	nNum	: UDINT;
END_VAR
IF nNum <= maxNumMover THEN
	aTrack[nNum] := ipTrack;
END_IF

SetStandardTrack := TRUE;
END_METHOD

METHOD UpdateMoverStatus : ST_MoverVisualisation
VAR
	nLogLineCnt		: UINT;
	nLogToDisplay	: UINT;
END_VAR
IF aMover[GVL_internal.nMoverIdToDisplay] = 0 THEN
	RETURN;
END_IF


GVL_internal.stMoverVisuData.nScrollBarMin := 0;
GVL_internal.stMoverVisuData.nScrollBarMax := MAX_LAST_LOGS - 10;


FOR nLogLineCnt := 1 TO 10 DO
	nLogToDisplay := nLogLineCnt + GVL_internal.stMoverVisuData.nScrollBarValue;
	nLogToDisplay := MIN(nLogToDisplay,MAX_LAST_LOGS);	

	GVL_internal.stMoverCmdLog[nLogLineCnt] := aMover[GVL_internal.nMoverIdToDisplay].GEtCommandLog(nLogToDisplay);
END_FOR
END_METHOD

METHOD PRIVATE UpdateTrackLog : ST_TrackVisualisation
VAR
	nLogLineCnt	  : UINT;
	nLogToDisplay : UINT;
END_VAR
IF aTrack[GVL_internal.nTrackIdToDisplay] = 0 THEN
	RETURN;
END_IF

GVL_internal.stTrackVisuData.nScrollBarMin := 0;
GVL_internal.stTrackVisuData.nScrollBarMax := MAX_LAST_LOGS - 10;

FOR nLogLineCnt := 1 TO 10 DO
	
	nLogToDisplay := nLogLineCnt + GVL_internal.stTrackVisuData.nScrollBarValue;
	nLogToDisplay := MIN(nLogToDisplay,MAX_LAST_LOGS);
		
	GVL_internal.stTrackCmdLog[nLogLineCnt] := aTrack[GVL_internal.nTrackIdToDisplay].GEtCommandLog(nLogToDisplay);
END_FOR
END_METHOD

END_FUNCTION_BLOCK

// XPlanarStandardFunctions/Visualization/Helper/VI_Background
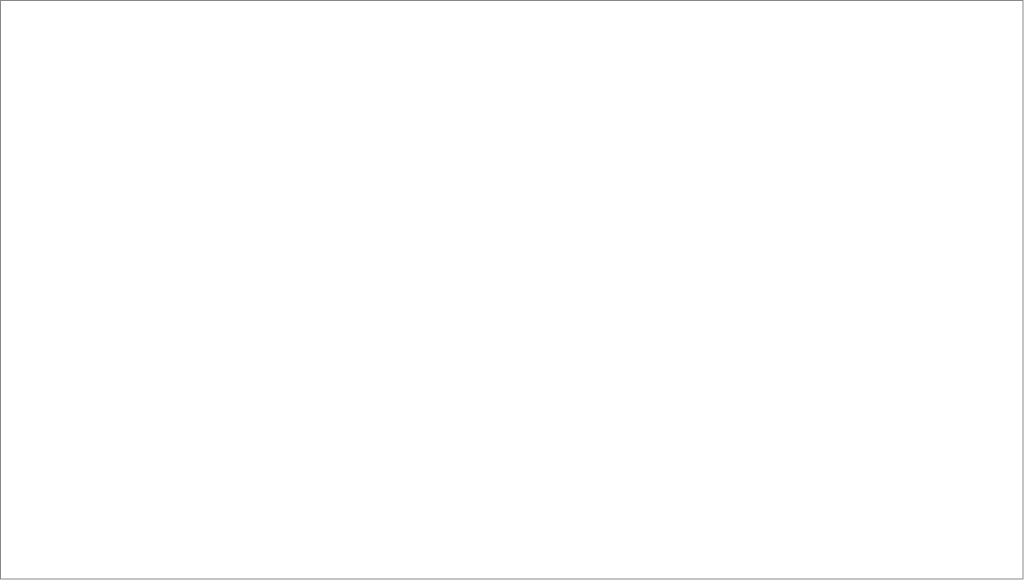
VISUALIZATION VI_Background  // 1024x580
    Rectangle (0,0 1024x580)
END_VISUALIZATION

// XPlanarStandardFunctions/Visualization/MoverLog/VI_MoverLogOverview
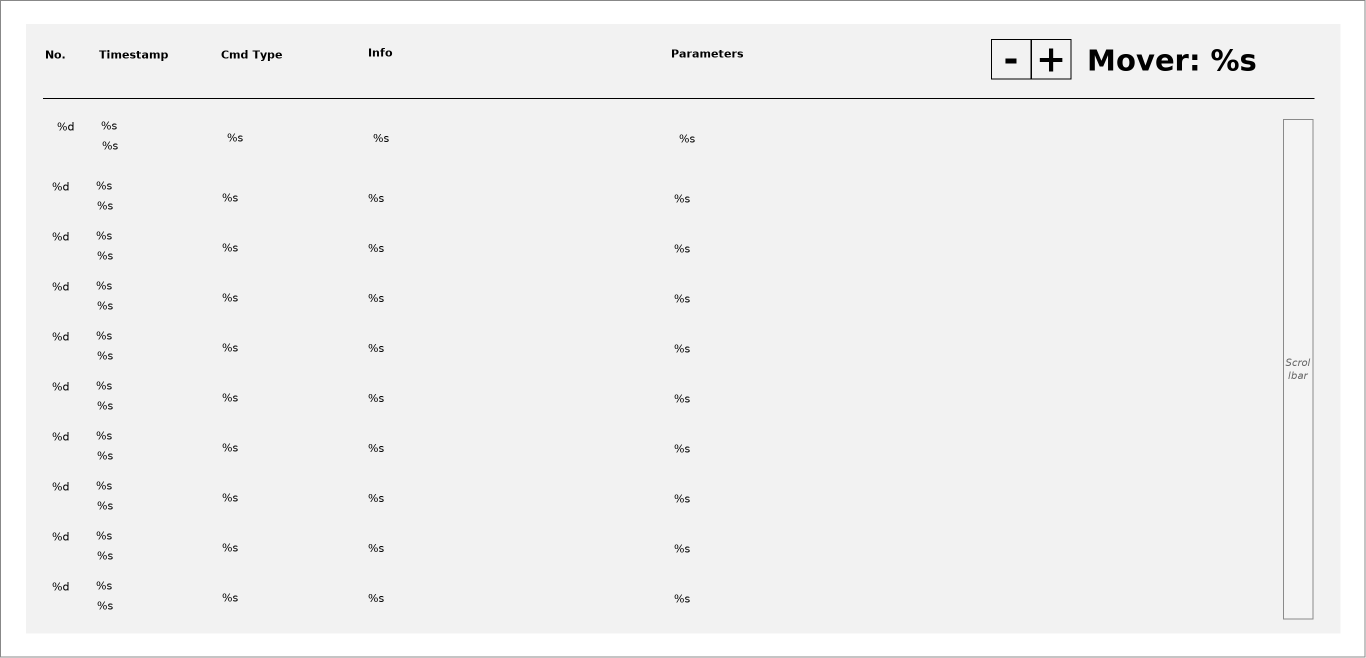
VISUALIZATION VI_MoverLogOverview  // 1366x658
    Rectangle (0,0 1368x657)
    Rectangle (26,24 1314x609)
    Rectangle (96,40 180x30), "Timestamp"
    Rectangle (42,40 44x30), "No."
    Frame (49,113 1230x50)
        shows VI_MoverLogOverview_Single(stCommandLog := GVL_internal.stMoverCmdLog[1])
    Frame (44,173 1230x50)
        shows VI_MoverLogOverview_Single(stCommandLog := GVL_internal.stMoverCmdLog[2])
    Frame (44,223 1230x50)
        shows VI_MoverLogOverview_Single(stCommandLog := GVL_internal.stMoverCmdLog[3])
    Frame (44,273 1230x50)
        shows VI_MoverLogOverview_Single(stCommandLog := GVL_internal.stMoverCmdLog[4])
    Frame (44,323 1230x50)
        shows VI_MoverLogOverview_Single(stCommandLog := GVL_internal.stMoverCmdLog[5])
    Frame (44,373 1230x50)
        shows VI_MoverLogOverview_Single(stCommandLog := GVL_internal.stMoverCmdLog[6])
    Frame (44,423 1230x50)
        shows VI_MoverLogOverview_Single(stCommandLog := GVL_internal.stMoverCmdLog[7])
    Frame (44,473 1230x50)
        shows VI_MoverLogOverview_Single(stCommandLog := GVL_internal.stMoverCmdLog[8])
    Frame (44,523 1230x50)
        shows VI_MoverLogOverview_Single(stCommandLog := GVL_internal.stMoverCmdLog[9])
    Frame (44,573 1230x50)
        shows VI_MoverLogOverview_Single(stCommandLog := GVL_internal.stMoverCmdLog[10])
    Rectangle (82,70 424x30)
    Line (43,98) (1314,98)
    Rectangle (218,40 77x30), "Cmd Type"
    Rectangle (668,39 180x30), "Parameters"
    Rectangle (1031,39 40x40), "+"
        tap GVL_internal.bNextMover
    Rectangle (991,39 40x40), "-"
        tap GVL_internal.bPreviousMover
    Rectangle (1084,41 223x39), "Mover: %s", text variable: GVL_internal.nMoverIdToDisplay
    Rectangle (365,38 180x30), "Info"
    Scrollbar (1283,119 30x500), invisible if: FALSE
        p3598130195: GVL_internal.stMoverVisuData.nScrollBarMin
        p2245068023: GVL_internal.stMoverVisuData.nScrollBarMax
        p1057716461: GVL_internal.stMoverVisuData.nScrollBarValue
END_VISUALIZATION

// XPlanarStandardFunctions/Visualization/MoverLog/VI_MoverLogOverview_Single
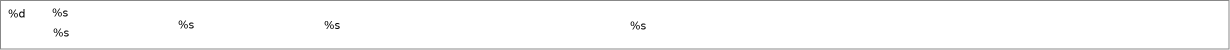
VISUALIZATION VI_MoverLogOverview_Single  // 1230x50
VAR_INPUT
	stCommandLog : ST_MoverCommandLog;
END_VAR
    Rectangle (0,0 1233x50)
    Rectangle (49,-12 180x50), "%s", text variable: stCommandLog.sTimeStampDate
    Rectangle (175,0 134x50), "%s", text variable: stCommandLog.sCommandType
    Rectangle (627,1 604x50), "%s", text variable: stCommandLog.sText
    Rectangle (5,-11 59x50), "%d", text variable: stCommandLog.nNo
    Rectangle (321,11 282x29), "%s", text variable: stCommandLog.sStation
    Rectangle (50,8 180x50), "%s", text variable: stCommandLog.sTimeStampTime
END_VISUALIZATION

// XPlanarStandardFunctions/Visualization/MoverLog/VI_MoverLogOverview_Single_1
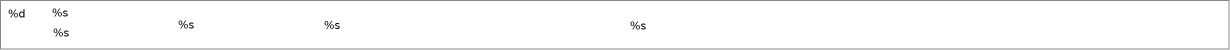
VISUALIZATION VI_MoverLogOverview_Single_1  // 1230x50
VAR_INPUT
	stCommandLog : ST_MoverCommandLog;
END_VAR
    Rectangle (0,0 1233x50)
    Rectangle (49,-12 180x50), "%s", text variable: stCommandLog.sTimeStampDate
    Rectangle (175,0 134x50), "%s", text variable: stCommandLog.sCommandType
    Rectangle (627,1 604x50), "%s", text variable: stCommandLog.sText
    Rectangle (5,-11 59x50), "%d", text variable: stCommandLog.nNo
    Rectangle (321,11 282x29), "%s", text variable: stCommandLog.sStation
    Rectangle (50,8 180x50), "%s", text variable: stCommandLog.sTimeStampTime
END_VISUALIZATION

// XPlanarStandardFunctions/Visualization/TrackLog/VI_TrackLogOverview
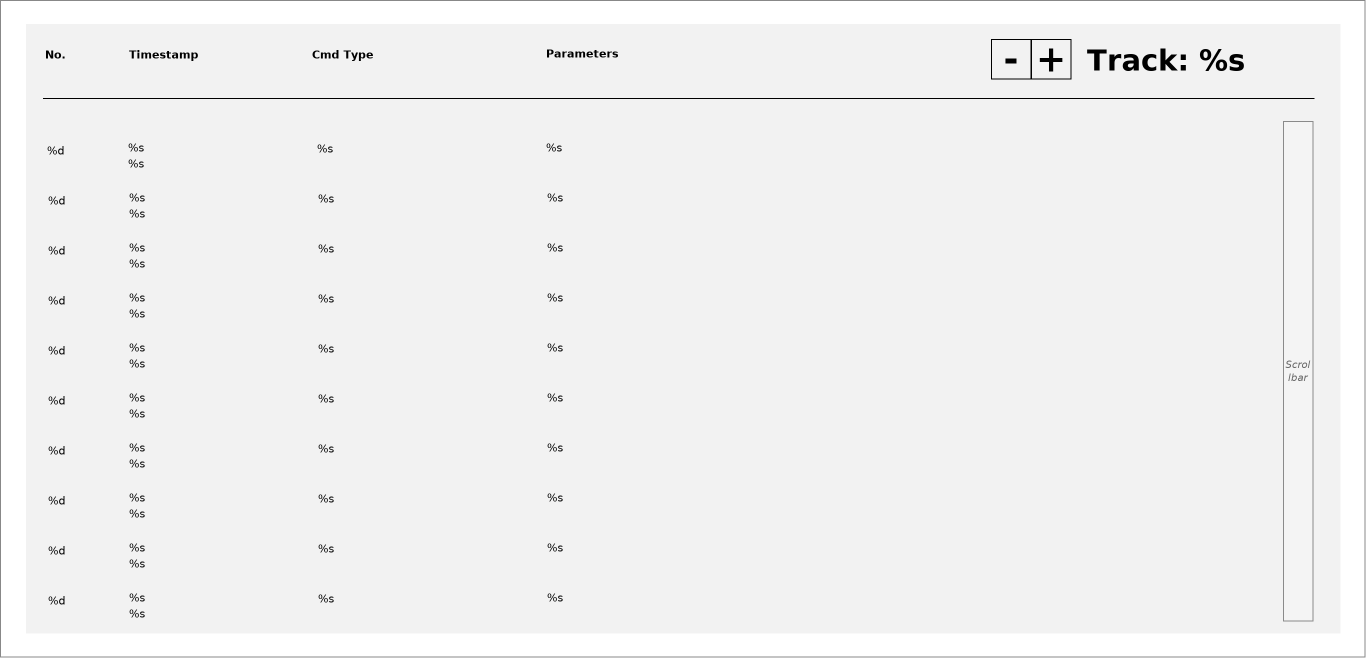
VISUALIZATION VI_TrackLogOverview  // 1366x658
    Rectangle (0,0 1368x657)
    Rectangle (26,24 1314x609)
    Rectangle (126,40 180x30), "Timestamp"
    Rectangle (42,40 44x30), "No."
    Frame (40,123 1230x50)
        shows VI_TrackLogOverview_Single(stCommandLog := GVL_internal.stTrackCmdLog[1])
    Frame (41,173 1230x50)
        shows VI_TrackLogOverview_Single(stCommandLog := GVL_internal.stTrackCmdLog[2])
    Frame (41,223 1230x50)
        shows VI_TrackLogOverview_Single(stCommandLog := GVL_internal.stTrackCmdLog[3])
    Frame (41,273 1230x50)
        shows VI_TrackLogOverview_Single(stCommandLog := GVL_internal.stTrackCmdLog[4])
    Frame (41,323 1230x50)
        shows VI_TrackLogOverview_Single(stCommandLog := GVL_internal.stTrackCmdLog[5])
    Frame (41,373 1230x50)
        shows VI_TrackLogOverview_Single(stCommandLog := GVL_internal.stTrackCmdLog[6])
    Frame (41,423 1230x50)
        shows VI_TrackLogOverview_Single(stCommandLog := GVL_internal.stTrackCmdLog[7])
    Frame (41,473 1230x50)
        shows VI_TrackLogOverview_Single(stCommandLog := GVL_internal.stTrackCmdLog[8])
    Frame (41,523 1230x50)
        shows VI_TrackLogOverview_Single(stCommandLog := GVL_internal.stTrackCmdLog[9])
    Frame (41,573 1230x50)
        shows VI_TrackLogOverview_Single(stCommandLog := GVL_internal.stTrackCmdLog[10])
    Rectangle (82,70 424x30)
    Line (43,98) (1314,98)
    Scrollbar (1283,121 30x500), invisible if: FALSE
        p3598130195: GVL_internal.stTrackVisuData.nScrollBarMin
        p2245068023: GVL_internal.stTrackVisuData.nScrollBarMax
        p1057716461: GVL_internal.stTrackVisuData.nScrollBarValue
    Rectangle (309,40 180x30), "Cmd Type"
    Rectangle (543,39 180x30), "Parameters"
    Rectangle (1031,39 40x40), "+"
        tap GVL_internal.bNextTrack
    Rectangle (991,39 40x40), "-"
        tap GVL_internal.bPreviousTrack
    Rectangle (1084,41 215x39), "Track: %s", text variable: GVL_internal.nTrackIdToDisplay
END_VISUALIZATION

// XPlanarStandardFunctions/Visualization/TrackLog/VI_TrackLogOverview_Single
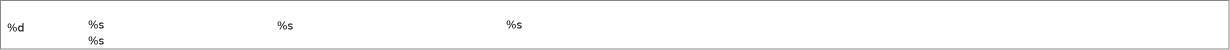
VISUALIZATION VI_TrackLogOverview_Single  // 1230x50
VAR_INPUT
	stCommandLog : ST_TrackCommandLog;
END_VAR
    Rectangle (0,0 1233x50)
    Rectangle (85,0 265x50), "%s", text variable: stCommandLog.sTimeStampDate
    Rectangle (274,1 199x50), "%s", text variable: stCommandLog.sCommandType
    Rectangle (503,0 513x50), "%s", text variable: stCommandLog.sText
    Rectangle (4,3 59x50), "%d", text variable: stCommandLog.nNo
    Rectangle (85,16 265x50), "%s", text variable: stCommandLog.sTimeStampTime
END_VISUALIZATION
